(* CODESYS project Tc3_XPlanarStandard.library
   Company: Beckhoff Automation GmbH
   DefaultNamespace: Tc3_XPlanarStandard
   Version: 3.3.2411.0
   Placeholder: Tc3_XPlanarStandard
   Title: Tc3_XPlanarStandard

Project tree, tasks and I/O mapping:
  libraries: Tc2_EtherCAT, * (Beckhoff Automation GmbH); Tc2_Math, * (Beckhoff Automation GmbH); Tc2_MC2, * (Beckhoff Automation GmbH); Tc2_Standard, * (Beckhoff Automation GmbH); Tc2_System, * (Beckhoff Automation GmbH); Tc2_Utilities, * (Beckhoff Automation GmbH); Tc3_EventLogger, * (Beckhoff Automation GmbH); Tc3_Mc3PlanarMotion, * (Beckhoff Automation GmbH); Tc3_Module, * (Beckhoff Automation GmbH); Tc3_Physics, * (Beckhoff Automation GmbH); Tc3_XPlanarUtility, * (Beckhoff Automation GmbH)
  BaseMover/
    ITFs/
      interface I_MoverBase: MoverID
  GeneralStandardFunctions/
    function ConvertToEventEntry [ST]
    function block FB_TcMoverMessage [ST]: AddError, AddInfo, SendMessage, SetSucceeded
    data type ST_ActualMotionParameters
  Version/
    global variables Global_Version
  XPlanarStandardFunctions/
    JoinClosestTrack/
      DUTs/
        data type ST_ErrorDetails
        data type ST_TrackDistance
        data type ST_TrackReachingTrial
      function block FB_JoinClosestTrack [ST]: AddTrack, AssignMover, ClearTracks, Locked, TracksCount, Execute
    MotionSystem/
      DUTs/
        data type E_MethodKeepAliveMotionSystem
        data type ST_CommandReturn
        data type ST_CommandReturnGearInPosOnTrack
        data type ST_CommandReturnGearInPosOnTrackWithMasterMover
        data type ST_CommandReturnInfo
        data type ST_MoverCheckInfo
      function block FB_XPlanarSystem [ST]: P_AddEnviromentToGroup, P_AddModuleToEnvironment, P_AddMoversToGroup, P_AddMoverToGroup, P_AddTracksToGroup, P_CheckValidMovers, P_DisableGroup, P_DisableMovers, P_DisableTracks, P_EnableGroup, P_EnableMovers, P_EnableTrack, P_EnableTracks, P_HaltSystem, P_LeaveTrack, P_PartActivatePosition, P_PartAllowEnable, P_PartForceDisable, P_PartForceEnable, P_PartInitialize, P_PartInitializeMulti, P_PartReset, P_RemoveEnviromentFromGroup, P_RemoveMoverFromGroup, P_RemoveMoversFromGroup, P_RemoveTracksFromGroup, P_ResetGroup, P_ResetMovers, P_ResetParts, P_ResetTracks, AddEnvironmentToGroup, AddModuleToEnvironment, AddMoversToGroup, AddMoverToGroup, AddTracksToGroup, CheckValidMovers, DisableGroup, DisableMovers, DisableTracks, EnableGroup, EnableMovers, EnableTrack, EnableTracks, HaltSystem, LeaveTrack, PartActivatePosition, PartAllowEnable, PartForceDisable, PartForceEnable, PartInitialize, PartInitializeMulti, PartReset, RemoveEnvironmentFromGroup, RemoveMoverFromGroup, RemoveMoversFromGroup, RemoveTracksFromGroup, ResetGroup, ResetMovers, ResetParts, ResetTracks, UtilityCheckForError, UtilityErrorReset, ccl_AddEnvironmentToGroup, ccl_AddModuleToEnvironment, ccl_AddMoversToGroup, ccl_AddMoverToGroup, ccl_AddTracksToGroup, ccl_CheckValidMovers, ccl_DisableGroup, ccl_DisableMovers, ccl_DisableTracks, ccl_EnableGroup, ccl_EnableMovers, ccl_EnableTrack, ccl_EnableTracks, ccl_HaltSystem, ccl_LeaveTrack, ccl_MethodKeepAlive, ccl_PartActivatePosition, ccl_PartAllowEnable, ccl_PartForceDisable, ccl_PartForceEnable, ccl_PartInitialize, ccl_PartInitializeMulti, ccl_PartReset, ccl_RemoveEnvironmentFromGroup, ccl_RemoveMoverFromGroup, ccl_RemoveMoversFromGroup, ccl_RemoveTracksFromGroup, ccl_ResetGroup, ccl_ResetMovers, ccl_ResetParts, ccl_ResetTracks, ResetStateVariables, Cycle, ipDriver, ipTcIoMover, P_IndexXPU, P_SystemInitialized, SetMoverStandard, SetTrackStandard, WriteParameter
      interface I_MotionSystem: P_AddEnviromentToGroup, P_AddModuleToEnvironment, P_AddMoversToGroup, P_AddMoverToGroup, P_AddTracksToGroup, P_CheckValidMovers, P_DisableGroup, P_DisableMovers, P_DisableTracks, P_EnableGroup, P_EnableMovers, P_EnableTrack, P_EnableTracks, P_HaltSystem, P_LeaveTrack, P_PartActivatePosition, P_PartAllowEnable, P_PartForceDisable, P_PartInitialize, P_PartInitializeMulti, P_PartReset, P_RemoveEnviromentFromGroup, P_RemoveMoverFromGroup, P_RemoveMoversFromGroup, P_RemoveTracksFromGroup, P_ResetGroup, P_ResetMovers, P_ResetParts, P_ResetTracks, AddEnvironmentToGroup, AddModuleToEnvironment, AddMoversToGroup, AddMoverToGroup, AddTracksToGroup, CheckValidMovers, DisableGroup, DisableMovers, DisableTracks, EnableGroup, EnableMovers, EnableTrack, EnableTracks, HaltSystem, LeaveTrack, PartActivatePosition, PartAllowEnable, PartForceDisable, PartInitialize, PartInitializeMulti, PartReset, RemoveEnvironmentFromGroup, RemoveMoverFromGroup, RemoveMoversFromGroup, RemoveTracksFromGroup, ResetGroup, ResetMovers, ResetParts, ResetTracks, UtilityCheckForError, UtilityErrorReset, Cycle, ipDriver, P_IndexXPU, P_SystemInitialized, SetMoverStandard, SetTrackStandard, WriteParameter
    Mover/
      BaseFunctions/
        function MoverVectorToPostionXYC [ST]
      DUTs/
        Log/
          data type E_MoverCommandType
          data type ST_GearInPosOnTrackMasterMoverParameterLog
          data type ST_GearInPosOnTrackParameterLog
          data type ST_JoinTrackLog
          data type ST_LeaveTrackInPositionLog
          data type ST_LeaveTrackLog
          data type ST_MoveOnTrackParameters
          data type ST_MoveOnTrackParametersLog
          data type ST_MoverCommand
          data type ST_MoverCommandLog
          data type ST_MoveToPositionExtParametersLog
          data type ST_MoveToPositionParametersLog
          data type ST_SetPositionParametersLog
        data type E_HaltDynamicsMode
        data type ST_CheckStartConditionFeedback
        data type ST_CheckStartConditionFeedbackExt
        data type ST_DynamicsVADJ
        data type ST_HaltDynamics
        data type ST_HaltParameter
        data type ST_TrackTableInfo
      Experimental/
        function block FB_MoverTarget [ST]: AddMover, AddPosition, Clear, MoversToTarget, P_ErrorWarningCode, P_Info, SetDynamics
        data type ST_MoverDistance
      ITFs/
      function block FB_XPlanarMoverStandard [ST]: P_DcTimeStamp, GetCommandLog, MoverCommandToString, UpdateCommandHistory, CheckStartConditions, GetCustomTrackID, GetDistanceToTrack, GetLastKnownCustomTrackID, MoveOnTrack, MoveToPosition, AddToGroup, AdoptTrackOrientation, Disable, DisableExternalSetpointGeneration, Enable, EnableExternalSetpointGeneration, GearInPosOnTrack, GetPositionOnCurrentPart, Halt, JoinTrack, LeaveTrack, LeaveTrackInPosition, MoveA, MoveB, MoveC, MoveOnTrackExt, MoveToPositionExt, MoveToPositionXYC, MoveZ, RemoveFromGroup, Reset, SetExternalSetpointValues, SetMoverPosition, CopyReturnStructure, CopyReturnStructureGearInPosOnTrack, CopyReturnStructureGearInPosOnTrackMasterMover, UpdateActualMotionParameter, P_AtRotationPoint, P_ClosestQuaterAngle, P_CRotationRestrictions, P_CustomTrackIdTable, P_HaltDynamics, P_IsMovingXY, P_IsPresent, P_IsQueuing, P_IsSetpointGeneratorActive, P_LastKnownTrackOID, P_RotationAngleModulo, P_SavedMoveOnTrackParameter, P_ZeroVelocityThreshold, P_AddToGroup, P_AdoptTrackOrientation, P_Disable, P_DisableExternalSetpointGeneration, P_Enable, P_EnableExternalSetpointGeneration, P_GearInPosOnTrack, P_GearInPosOnTrackMasterMover, P_Halt, P_JoinTrack, P_LeaveTrack, P_LeaveTrackInPosition, P_MoveA, P_MoveB, P_MoveC, P_MoveOnTrack, P_MoveOnTrackExt, P_MoveToPosition, P_MoveToPositionExt, P_MoveToPositionXYC, P_MoveZ, P_RemoveFromGroup, P_Reset, P_SetMoverPosition, P_ActPosition, P_ActVelocity, P_Busy, P_CommandMode, P_Error, P_ErrorCode, P_ErrorID, P_Id, P_InGroup, P_MoverOid, P_MoverRef, P_PhysicalAreaID, P_SetAcceleration, P_SetOnTrack, P_SetPosition, P_SetVelocity, P_State, P_TrackId, Cycle
      interface I_XPlanarMoverStandard: P_DcTimeStamp, CheckStartConditions, GetCustomTrackID, GetDistanceToTrack, GetLastKnownCustomTrackID, MoveOnTrack, MoveToPosition, AddToGroup, AdoptTrackOrientation, Disable, DisableExternalSetpointGeneration, Enable, EnableExternalSetpointGeneration, GearInPosOnTrack, GetCommandLog, GetPositionOnCurrentPart, Halt, JoinTrack, LeaveTrack, LeaveTrackInPosition, MoveA, MoveB, MoveC, MoveOnTrackExt, MoveToPositionExt, MoveToPositionXYC, MoveZ, RemoveFromGroup, Reset, SetExternalSetpointValues, SetMoverPosition, P_AtRotationPoint, P_ClosestQuaterAngle, P_CRotationRestrictions, P_CustomTrackIdTable, P_HaltDynamics, P_IsMovingXY, P_IsPresent, P_IsQueuing, P_IsSetpointGeneratorActive, P_LastKnownTrackOID, P_RotationAngleModulo, P_SavedMoveOnTrackParameter, P_ZeroVelocityThreshold, P_AddToGroup, P_AdoptTrackOrientation, P_Disable, P_DisableExternalSetpointGeneration, P_Enable, P_EnableExternalSetpointGeneration, P_GearInPosOnTrack, P_GearInPosOnTrackMasterMover, P_Halt, P_JoinTrack, P_LeaveTrack, P_LeaveTrackInPosition, P_MoveA, P_MoveB, P_MoveC, P_MoveOnTrack, P_MoveOnTrackExt, P_MoveToPosition, P_MoveToPositionExt, P_MoveToPositionXYC, P_MoveZ, P_RemoveFromGroup, P_Reset, P_SetMoverPosition, P_ActPosition, P_ActVelocity, P_Busy, P_CommandMode, P_Error, P_ErrorCode, P_ErrorID, P_Id, P_InGroup, P_MoverOid, P_MoverRef, P_PhysicalAreaID, P_SetAcceleration, P_SetOnTrack, P_SetPosition, P_SetVelocity, P_State, P_TrackId, Cycle
    MoverQueue/
      DUTs/
        data type ST_MoverOnTrack
      function block FB_MoverQueue [ST]: Clear, Dequeue, Enqueue, Count, Item
      interface I_MoverQueue: Clear, Dequeue, Enqueue, Count, Item
    Station/
      DUTs/
        data type eSortingDirection
        data type eSortingMode
        data type ST_List
        data type ST_MoverInList
      function block FB_List [ST]: P_eSortingMode, P_fSortingOrigin, P_nNumberInList, P_nResult, P_nSortingMode, P_sMessage, P_SortingMode, AddMover, AddTrack, ClearList, ClearTrackOrder, CopyList, GetMoverIndexInListPosition, GetMoverInListPosition, P_FirstInList, P_Message, P_MoverList, P_NumberInList, P_Result, P_SortingDirection, P_SortingOrigin, P_TrackBuiltInfo, RemoveFirstInList, RemoveFromList, SortList
      interface I_List: P_eSortingMode, P_fSortingOrigin, P_nNumberInList, P_nResult, P_nSortingMode, P_sMessage, AddMover, AddTrack, ClearList, ClearTrackOrder, GetMoverIndexInListPosition, GetMoverInListPosition, P_FirstInList, P_Message, P_MoverList, P_NumberInList, P_Result, P_SortingMode, P_SortingOrigin, P_TrackBuiltInfo, RemoveFirstInList, RemoveFromList, SortList
    Track/
      DUTs/
        data type E_MethodKeepAliveTrack
        data type E_PointOption
        data type E_PointType
        data type E_TrackCommandType
        data type ST_BuildTrackParameterLog
        data type ST_CutomTrackID
        data type ST_LoggingVisu
        data type ST_StartEndAtTrackParameterLog
        data type ST_TrackAppendCircleParameterLog
        data type ST_TrackAppendLineParameterLog
        data type ST_TrackAppendPointParameterLog
        data type ST_TrackBuildParameter
        data type ST_TrackBuiltInfo
        data type ST_TrackCommand
        data type ST_TrackCommandLog
        data type ST_TrackInfo
        data type ST_TrackPoint
        data type ST_TrackTable
      function block FB_CustomTrackIdTable [ST]: Clear, P_TabelData, SetTrack
      function block FB_TrackStandard [ST]: ccl_BuildTrack, ccl_BuildTrackAdv, ccl_BuildTrackExt, ccl_MethodKeepAlive, CopyReturnStructure, ref, GetCommandLog, TrackCommandToString, UpdateCommandHistory, P_AddToGroup, P_AppendCircle, P_AppendLine, P_AppendPoint, P_BuildTrack, P_BuildTrackAdvanced, P_BuildTrackAdvanced_Check, P_BuildTrackAdvancedInfoText, P_BuildTrackExt, P_BuildTrackExtInfoText, P_Clear, P_CloseLoop, P_Disable, P_Enable, P_EndAtTrack, P_RemoveFromGroup, P_Reset, P_StartFromTrack, AddToGroup, AppendCircle, AppendLine, AppendPoint, BuildTrack, BuildTrackAdvanced, BuildTrackExt, Clear, CloseLoop, cycle, Disable, Enable, EndAtTrack, EndAtTrackAdv, GetLength, GetMoverPositionAt, GetTrackPositionAt, GetTrackPositionAt_XY, P_GroupOID, P_Info, P_MoverCountOnTrack, P_MovingMoverCount, P_OID, P_OperationMode, P_State, P_TrackBuiltInfo, P_TrackRef, RemoveFromGroup, Reset, StartFromTrack, StartFromTrackAdv
      function block FB_TrackTable [ST]: AddPoint, CheckTrackTable, ClearTrackTable, P_BuildlParameter, P_CloseTheLoop, P_EndAtTrack, P_InfoText, P_NumberOfPointsInTable, P_StartFromTrack, P_Table, P_TrackCheckImplausibleTableIndex, P_TrackTableCheckResult
      function block FB_TrackTableAdvanced [ST]: AddPoint, CheckPoint, CheckTrackTable, ClearTrackTable, P_BuildlParameter, P_CloseTheLoop, P_EndAtTrack, P_EndAtTrackOptions, P_InfoText, P_NumberOfPointsInTable, P_StartFromTrack, P_StartFromTrackOptions, P_Table, P_TrackCheckImplausibleTableIndex, P_TrackTableCheckResult
      interface I_CustomTrackIndexTable: P_TabelData
      interface I_TrackStandard: P_AddToGroup, P_AppendCircle, P_AppendLine, P_AppendPoint, P_BuildTrack, P_BuildTrackAdvanced, P_BuildTrackAdvanced_Check, P_BuildTrackAdvancedInfoText, P_BuildTrackExt, P_Clear, P_CloseLoop, P_Disable, P_Enable, P_EndAtTrack, P_RemoveFromGroup, P_Reset, P_StartFromTrack, AddToGroup, AppendCircle, AppendLine, AppendPoint, BuildTrack, BuildTrackAdvanced, BuildTrackExt, Clear, CloseLoop, Cycle, Disable, Enable, GetCommandLog, GetLength, GetMoverPositionAt, GetTrackPositionAt, GetTrackPositionAt_XY, P_GroupOID, P_Info, P_MoverCountOnTrack, P_MovingMoverCount, P_OID, P_OperationMode, P_State, P_TrackRef, ref, RemoveFromGroup, Reset
    Visualization/
      DUTs/
        data type ST_MoverVisualisation
        data type ST_TrackVisualisation
      Helper/
        visualisation VI_Background
      MoverLog/
        visualisation VI_MoverLogOverview
        visualisation VI_MoverLogOverview_Single
        visualisation VI_MoverLogOverview_Single_1
      TrackLog/
        visualisation VI_TrackLogOverview
        visualisation VI_TrackLogOverview_Single
      function block FB_XPlanarVisuDiag [ST]: Cycle, SetStandardMover, SetStandardTrack, UpdateMoverStatus, UpdateTrackLog
  text list GlobalTextList
  global variables GVL_internal
  global variables GVL_Tc3XPlanarStandard
  global variables Params_XPlanar
*)

// GeneralStandardFunctions/ST_ActualMotionParameters
TYPE ST_ActualMotionParameters :
STRUCT
	Position			: MoverVector;
	fSetTrackPosition	: LREAL;
	nTrackOid 			: OTCID;
	sTrackName 			: STRING(80);
	fSetVelo			: LREAL;
	fSetAcc				: LREAL;	
END_STRUCT
END_TYPE

// XPlanarStandardFunctions/JoinClosestTrack/DUTs/ST_ErrorDetails
TYPE ST_ErrorDetails :
STRUCT
	TrackOID	: OTCID;			// Track object ID
	ErrorID		: UDINT;			// Error ID
	objectInfo	: PlanarObjectInfo;	// Object causing error
END_STRUCT
END_TYPE

// XPlanarStandardFunctions/JoinClosestTrack/DUTs/ST_TrackDistance
TYPE ST_TrackDistance :
STRUCT
	TrackOID		: OTCID;			// Track object ID
	Index			: UDINT;			// Index in Track list
	CurrentLocation	: MoverVector;		// Current position of the Mover
	PositionOnTrack	: LREAL;			// Arc position on Track after JoinTrack() command
	IsPossibleTrack	: BOOL;				// Joining this track is possible
	ErrorID			: UDINT;			// Error ID making track impossible to join
	objectInfo		: PlanarObjectInfo;	// Object causing collision
	TargetLocation	: MoverVector;		// Mover position after JoinTrack() command
	Distance		: LREAL;			// Absolute distance [mm]
END_STRUCT
END_TYPE

// XPlanarStandardFunctions/JoinClosestTrack/DUTs/ST_TrackReachingTrial
TYPE ST_TrackReachingTrial :
STRUCT
	TrackInfo	: ST_TrackDistance;	// Track distance info
	Done		: BOOL;				// JoinTrack operation has succeed
	Busy		: BOOL;				// JoinTrack operation is busy
	Error		: BOOL;				// JoinTrack operation has failed
	ErrorID		: UDINT;			// Error ID at failure
	objectInfo	: PlanarObjectInfo;	// Object causing collision
END_STRUCT
END_TYPE

// XPlanarStandardFunctions/MotionSystem/DUTs/E_MethodKeepAliveMotionSystem
{attribute 'qualified_only'}
{attribute 'strict'}
TYPE E_MethodKeepAliveMotionSystem :
(
	eIdle := 0,
	eAddMoverToGroup,
	eAddMoversToGroup,
	eAddEnvironmentToGroup,
	eAddTracksToGroup,
	eDisableGroup,
	eDisableMovers,
	eDisableSystem,
	eEnableGroup,
	eEnableMovers,
	eEnableSystem,
	eEnableTrack,
	eEnableTracks,
	eDisableTracks,
	eHaltSystem,
	eLeaveTrack,
	eRemoveMoverFromGroup,
	eRemoveMoversFromGroup,
	eRemoveEnvironmentFromGroup,
	eRemoveTracksFromGroup,
	eResetGroup,
	eResetTracks,
	eResetMovers,
	eResetSystem,
	eError,
	eAddModuleToEnvironment,
	eCheckValidMovers,
	ePartInitialize,
	ePartInitializeMulti,
	ePartActivatePosition,
	ePartForceDisable,
	ePartForceEnable,
	ePartAllowEnable,
	ePartReset,
	eResetParts
);
END_TYPE

// XPlanarStandardFunctions/MotionSystem/DUTs/ST_CommandReturn
TYPE ST_CommandReturn :
STRUCT
	Done 	: BOOL;
	Busy 	: BOOL;
	Aborted	: BOOL;
	Active 	: BOOL;
	Error	: BOOL;
	ErrorID	: UDINT;
	stInfo 	: ST_CommandReturnInfo;
END_STRUCT
END_TYPE

// XPlanarStandardFunctions/MotionSystem/DUTs/ST_CommandReturnGearInPosOnTrack
TYPE ST_CommandReturnGearInPosOnTrack :
STRUCT
//	Done 	: BOOL;
	Busy 	: BOOL;
	Aborted	: BOOL;
	Active 	: BOOL;
	Error	: BOOL;
	ErrorID	: UDINT;
	stInfo 	: ST_CommandReturnInfo;
	inSync	: BOOL;
END_STRUCT
END_TYPE

// XPlanarStandardFunctions/MotionSystem/DUTs/ST_CommandReturnGearInPosOnTrackWithMasterMover
TYPE ST_CommandReturnGearInPosOnTrackWithMasterMover :
STRUCT
//	Done 	: BOOL;
	Busy 	: BOOL;
	Aborted	: BOOL;
	Active 	: BOOL;
	Error	: BOOL;
	ErrorID	: UDINT;
	stInfo 	: ST_CommandReturnInfo;
	inSync	: BOOL;
END_STRUCT
END_TYPE

// XPlanarStandardFunctions/MotionSystem/DUTs/ST_CommandReturnInfo
TYPE ST_CommandReturnInfo :
STRUCT
	nObjectType : UDINT;
	nObjectID 	: UDINT;
END_STRUCT
END_TYPE

// XPlanarStandardFunctions/MotionSystem/DUTs/ST_MoverCheckInfo
TYPE ST_MoverCheckInfo :
STRUCT
	bDone				: BOOL;	
	bAllMoversValid		: BOOL;
	bMoverLost			: BOOL;
	nValidMoverCount	: UDINT;	

END_STRUCT
END_TYPE

// XPlanarStandardFunctions/Mover/DUTs/Log/E_MoverCommandType
TYPE E_MoverCommandType :
(
	eMoverCommand_eNoCommand 			:= 0,
	eMoverCommand_eMoveAbs,
	eMoverCommand_eMoveModOnTrack,
	eMoverCommand_eMoveModOnTrackExt,		
	eMoverCommand_eMoveRel,			
	eMoverCommand_eHalt, 			
	eMoverCommand_eGearIn, 			
	eMoverCommand_eDynamicsChange, 		
	eMoverCommand_eGapChange, 		
	eMoverCommand_eSuperImposed, 	
	eMoverCommand_eCamInInstant, 	
	eMoverCommand_eCamInTwoTables, 	
	eMoverCommand_eCamOut, 			
	eMoverCommand_eReset, 			
	eMoverCommand_eEnable,			
	eMoverCommand_eDisable,			
	eMoverCommand_eAddMoverToGroup,	
	eMoverCommand_eRemoveMoverFromGroup,	
	eMoverCommand_eMoveAbsDone,		
	eMoverCommand_eMoveModDone,		
	eMoverCommand_eMoveRelDone,			
	eMoverCommand_eHaltCa,				
	eMoverCommand_eHaltCaDone,			
	eMoverCommand_eMoveAbsQueueing,	
	eMoverCommand_eMoveModQueueing,		
	eMoverCommand_eMoveRelQueueing,		
	eMoverCommand_eGearInInSync,		
	eMoverCommand_eGearOutOfSync,	
	eMoverCommand_eJoinTrack,			
	eMoverCommand_eLeaveTrack,		
	eMoverCommand_eLeaveTrackInPosition,	
	eMoverCommand_eMoveToPosition,		
	eMoverCommand_eMoveToPositionXYC,	
	eMoverCommand_eMoveToPositionExt,	
	eMoverCommand_eMoveZ,
	eMoverCommand_eMoveA,
	eMoverCommand_eMoveB,
	eMoverCommand_eMoveC,
	eMoverCommand_eEnableExternalSetPos,
	eMoverCommand_eDisableExternalSetPos,
	eMoverCommand_eCheckStartConditions,
	eMoverCommand_eAdoptTrackOrientation,
	eMoverCommand_eGearInPosOnTrack,
	eMoverCommand_eGearInPosOnTrackMasterMover,
	eMoverCommand_eSetPosition 	
	
	
);
END_TYPE

// XPlanarStandardFunctions/Mover/DUTs/Log/ST_GearInPosOnTrackMasterMoverParameterLog
TYPE ST_GearInPosOnTrackMasterMoverParameterLog :
STRUCT
	
	MasterMover			: UDINT;
	MasterSyncPos		: LREAL;
	TrackMasterSyncPos	: UDINT;
	SlaveSyncPos		: LREAL;
	TrackSlaveSyncPos	: UDINT;
	
	TrackTrailSize		: UDINT;	
	
	Velocity  			: LREAL;
	Acceleration		: LREAL;
	Deceleration		: LREAL;
	Jerk  				: LREAL;
	Gap					: LREAL;

	moduloToleranceMasterSyncPosition	: LREAL;
	directionMasterSyncPosition			: DINT;
	inSyncToleranceDistance				: LREAL;
	moduloToleranceSlaveSyncPosition	: LREAL;
	
	allowedSlaveSyncDirections			: DINT;
	directionSlaveSyncPosition			: DINT;
	
	followMover							: BOOL;
	
	
	

		
END_STRUCT
END_TYPE

// XPlanarStandardFunctions/Mover/DUTs/Log/ST_GearInPosOnTrackParameterLog
TYPE ST_GearInPosOnTrackParameterLog :
STRUCT
	
	MasterSyncPos	: LREAL;
	SlaveSyncPos	: LREAL;
	Velocity  		: LREAL;
	Acceleration	: LREAL;
	Deceleration	: LREAL;
	Jerk  			: LREAL;
	Gap				: LREAL;

	Track			: UDINT;
	TrackTrailSize	: UDINT;
	
	allowedSlaveSyncDirections	: Tc3_Mc3PlanarMotion.MC_SYNC_DIRECTIONS;
	directionSlaveSyncPosition  : Tc3_Mc3PlanarMotion.MC_Direction;
	
	inSyncToleranceDistance				: LREAL;
	moduloToleranceSlaveSyncPosition	: LREAL;
	
		
END_STRUCT
END_TYPE

// XPlanarStandardFunctions/Mover/DUTs/Log/ST_JoinTrackLog
TYPE ST_JoinTrackLog :
STRUCT
	nTargetTrack 		: OTCID;
	fVelo				: LREAL;		
	fAcc				: LREAL;
	fJerk				: LREAL;
END_STRUCT
END_TYPE

// XPlanarStandardFunctions/Mover/DUTs/Log/ST_LeaveTrackInPositionLog
TYPE ST_LeaveTrackInPositionLog :
STRUCT
	fPositionX			: LREAL;		
	fPositionY			: LREAL;		
	fPositionC			: LREAL;		
END_STRUCT
END_TYPE

// XPlanarStandardFunctions/Mover/DUTs/Log/ST_LeaveTrackLog
TYPE ST_LeaveTrackLog :
STRUCT
	fPositionX			: LREAL;		
	fPositionY			: LREAL;		
	fPositionC			: LREAL;		
	fVelo				: LREAL;		
	fAcc				: LREAL;
	fDec				: LREAL;
	fJerk				: LREAL;
END_STRUCT
END_TYPE

// XPlanarStandardFunctions/Mover/DUTs/Log/ST_MoveOnTrackParameters
TYPE ST_MoveOnTrackParameters:
STRUCT
	
	fTrackPosition	 	: LREAL;
	fVelo				: LREAL;	
	ipTrack				: I_TrackStandard;
	fAcc				: LREAL;
	fDec				: LREAL;
	fJerk				: LREAL;
	fGap				: LREAL;
	direction			: Tc3_Mc3PlanarMotion.MC_DIRECTION;
	
END_STRUCT
END_TYPE

// XPlanarStandardFunctions/Mover/DUTs/Log/ST_MoveOnTrackParametersLog
TYPE ST_MoveOnTrackParametersLog:
STRUCT
	
	fTargetPosition 	: LREAL;
	fVelo				: LREAL;	
	nTargetTrackOid		: OTCID;
	sTargetTrack		: STRING(80);
	nTargetTrackID		: UDINT;
	fAcc				: LREAL;
	fDec				: LREAL;
	fJerk				: LREAL;
	fGap				: LREAL;
	
END_STRUCT
END_TYPE

// XPlanarStandardFunctions/Mover/DUTs/Log/ST_MoverCommand
TYPE ST_MoverCommand : //structure for storing a list of commands to the mover 
STRUCT
	sStation				: STRING;	// Station Name that give a move command
	eCommandType 			: E_MoverCommandType; // what command was done
	
	stActualParameter			: ST_ActualMotionParameters;
//	stActualMasterParameter	: ST_ActualMotionParameters;
//	stGearInParameter		: ST_GearInParametersLog;
//	stMoveAbsoluteParameter	: ST_MoveAbsoluteParametersLog;
//	stMoveRelativeParameter	: ST_MoveRelativeParametersLog;
	stMoveOnTrackParameter					: ST_MoveOnTrackParametersLog;	
	stMoveOnTrackParameterExt				: ST_MoveOnTrackParametersLog;	
	stGearInPosOnTrackParameter				: ST_GearInPosOnTrackParameterLog;
	stGearInPosOnTrackMasterMoverParameter	: ST_GearInPosOnTrackMasteRMoverParameterLog;
	stMoveToPosition						: ST_MoveToPositionParametersLog;
	stMoveToPositionXYC						: ST_MoveToPositionParametersLog;
	stMoveToPositionExt						: ST_MoveToPositionExtParametersLog;	
 	stHaltParameter							: ST_HaltParameter;
	stJoinTrackParameter					: ST_JoinTrackLog;
	stLeaveTrackParameter					: ST_LeaveTrackLog;
	stLeaveTrackInPositionParameter			: ST_LeaveTrackInPositionLog;
	stSetPosition							: ST_SetPositionParametersLog;

	
	sText 					: STRING(255); 
	stTimeStamp 			: STRING ; //dcTimestampTime can be decoded later 
END_STRUCT
END_TYPE

// XPlanarStandardFunctions/Mover/DUTs/Log/ST_MoverCommandLog
TYPE ST_MoverCommandLog :
STRUCT
	nNo				: INT;
	sTimeStamp		: STRING;	
	sTimeStampDate	: STRING;
	sTimeStampTime	: STRING;	
	sStation		: STRING;
	sCommandType	: STRING;
	sText			: STRING(255);
END_STRUCT
END_TYPE

// XPlanarStandardFunctions/Mover/DUTs/Log/ST_MoveToPositionExtParametersLog
TYPE ST_MoveToPositionExtParametersLog:
STRUCT
	fVelo						: LREAL;	

	fTargetPositionX 			: LREAL;
	fTargetPositionY 			: LREAL;
	fTargetPositionC 			: LREAL;
	
	fAcc						: LREAL;
	fDec						: LREAL;
	fJerk						: LREAL;
	
	stMoveToPositionOptions		: ST_MoveToPositionOptions;
END_STRUCT
END_TYPE

// XPlanarStandardFunctions/Mover/DUTs/Log/ST_MoveToPositionParametersLog
TYPE ST_MoveToPositionParametersLog:
STRUCT


	fVelo				: LREAL;	

	fTargetPositionX 	: LREAL;
	fTargetPositionY 	: LREAL;
	fTargetPositionC 	: LREAL;
	
	fAcc				: LREAL;
	fDec				: LREAL;
	fJerk				: LREAL;	
	
	
END_STRUCT
END_TYPE

// XPlanarStandardFunctions/Mover/DUTs/Log/ST_SetPositionParametersLog
TYPE ST_SetPositionParametersLog:
STRUCT
	fPositionX 	: LREAL;
	fPositionY 	: LREAL;
	fPositionC 	: LREAL;
END_STRUCT
END_TYPE

// XPlanarStandardFunctions/Mover/DUTs/E_HaltDynamicsMode
{attribute 'qualified_only'}
{attribute 'strict'}
TYPE E_HaltDynamicsMode :
(
	AxisX_AxisY_CoordinatedOnPath 	:= 0,
	AxisX_AxisY_Separately			:= 1
);
END_TYPE

// XPlanarStandardFunctions/Mover/DUTs/ST_CheckStartConditionFeedback
TYPE ST_CheckStartConditionFeedback :
STRUCT

	nMoverID					: UINT;
	bPositionOK					: BOOL;	
	bPositionXLimitExceeded		: BOOL;
	bPositionYLimitExceeded		: BOOL;
	bAngleLimitExceeded			: BOOL;
	fCurrentAngleDeviation		: LREAL;
	fCurrentPositionDeviationX	: LREAL;
	fCurrentPositionDeviationY	: LREAL;	
	
END_STRUCT
END_TYPE

// XPlanarStandardFunctions/Mover/DUTs/ST_CheckStartConditionFeedbackExt
TYPE ST_CheckStartConditionFeedbackExt :
STRUCT

	nMoverID					: UINT;
	bPositionOK					: BOOL;	
	bFeedbackInvalid			: BOOL;
	bPositionXLimitExceeded		: BOOL;
	bPositionYLimitExceeded		: BOOL;
	bAngleLimitExceeded			: BOOL;
	fCurrentAngleDeviation		: LREAL;
	fCurrentPositionDeviationX	: LREAL;
	fCurrentPositionDeviationY	: LREAL;	
	
END_STRUCT
END_TYPE

// XPlanarStandardFunctions/Mover/DUTs/ST_DynamicsVADJ
TYPE ST_DynamicsVADJ :
STRUCT
	fVelocity		: LREAL;
	fAcceleration	: LREAL;
	fDeceleration	: LREAL;
	fJerk			: LREAL;	
END_STRUCT
END_TYPE

// XPlanarStandardFunctions/Mover/DUTs/ST_HaltDynamics
TYPE ST_HaltDynamics :
STRUCT
	
	PathXY		: ST_DynamicsVADJ;
	AxisX		: ST_DynamicsVADJ;
	AxisY		: ST_DynamicsVADJ;
	AxisZ		: ST_DynamicsVADJ;
	AxisA		: ST_DynamicsVADJ;
	AxisB		: ST_DynamicsVADJ;
	AxisC		: ST_DynamicsVADJ;	
	
	Mode		: E_HaltDynamicsMode;

END_STRUCT
END_TYPE

// XPlanarStandardFunctions/Mover/DUTs/ST_HaltParameter
TYPE ST_HaltParameter :
STRUCT
	
	fDeceleration_XY	: LREAL;
	fJerk_XY			: LREAL; 
	fDeceleration_A		: LREAL;
	fJerk_A				: LREAL; 
	fDeceleration_B		: LREAL;
	fJerk_B				: LREAL; 		
	fDeceleration_C		: LREAL;
	fJerk_C				: LREAL; 	
	
END_STRUCT
END_TYPE

// XPlanarStandardFunctions/Mover/DUTs/ST_TrackTableInfo
TYPE ST_TrackTableInfo :
STRUCT
	nTrackOID	: UDINT;
	nTrackID	: UDINT;	
END_STRUCT
END_TYPE

// XPlanarStandardFunctions/Mover/Experimental/ST_MoverDistance
{attribute 'hide'}
TYPE ST_MoverDistance :
STRUCT
	nPositionIndex	: UDINT;
	fDistance		: LREAL;
END_STRUCT
END_TYPE

// XPlanarStandardFunctions/MoverQueue/DUTs/ST_MoverOnTrack
TYPE ST_MoverOnTrack :
STRUCT
	ID			: UDINT;	// Mover ID
	MoverOID	: OTCID;	// Mover object ID
	PosOnTrack	: LREAL;	// Position on track
END_STRUCT
END_TYPE

// XPlanarStandardFunctions/Station/DUTs/eSortingDirection
TYPE eSortingDirection :
(
	ascending  := 0,
	descending := 1
);
END_TYPE

// XPlanarStandardFunctions/Station/DUTs/eSortingMode

TYPE eSortingMode :
(
	descending := 0,
	ascending  := 1
);
END_TYPE

// XPlanarStandardFunctions/Station/DUTs/ST_List
TYPE ST_List :
STRUCT
	nNumInList		: INT;
	//aMoverList 		: ARRAY[1..GVL_ListParameter.gcnMaxNumInList] OF I_XPlanarMoverStandard; 
	aMoverList 		: ARRAY[1..maxNumMover] OF I_XPlanarMoverStandard;
	
END_STRUCT
END_TYPE

// XPlanarStandardFunctions/Station/DUTs/ST_MoverInList
TYPE ST_MoverInList :
STRUCT
	nMoverIndex		 	: UDINT;
	nMoverPosition 		: LREAL;
	nMoverTrackOID 		: UDINT;	
END_STRUCT
END_TYPE

// XPlanarStandardFunctions/Track/DUTs/E_MethodKeepAliveTrack
{attribute 'qualified_only'}
{attribute 'strict'}
TYPE E_MethodKeepAliveTrack :
(
	eIdle          := 0,
	eBuildTrack    := 1,
	eBuildTrackExt := 2,
	eBuildTrackAdv := 3,
	eError
);
END_TYPE

// XPlanarStandardFunctions/Track/DUTs/E_PointOption
{attribute 'qualified_only'}
{attribute 'strict'}
TYPE E_PointOption :
(
	none,
	Circle_Clockwise,
	Circle_CounterClockwise
);
END_TYPE

// XPlanarStandardFunctions/Track/DUTs/E_PointType
{attribute 'qualified_only'}
{attribute 'strict'}
TYPE E_PointType :
(
	none,
	Point,
	Line_Start,
	Line_End,
	Circle_Start,
	Circle_Center,
	Circle_End
	
);
END_TYPE

// XPlanarStandardFunctions/Track/DUTs/E_TrackCommandType
TYPE E_TrackCommandType :
(
	eTrackCommand_eNoCommand 			:= 0,
	eTrackCommand_eEnable				:= 1,
	eTrackCommand_eDisable 				:= 2,
	eTrackCommand_eAppendLine 			:= 3,
	eTrackCommand_eCloseLoop			:= 4,
	eTrackCommand_eStartFromTrack		:= 5,	
	eTrackCommand_eEndAtTrack			:= 6,
	eTrackCommand_eAddToGroup			:= 7,
	eTrackCommand_eRemoveFromGroup		:= 8,
	eTrackCommand_eAppendPoint			:= 9,
	eTrackCommand_eAppendCircle			:= 10,
	eTrackCommand_eBuildTrack			:= 11,	
	eTrackCommand_eReset				:= 12,
	eTrackCommand_eClear				:= 13,
	eTrackCommand_eStartFromTrackAdv	:= 14,
	eTrackCommand_eAppendPointAdv		:= 15,
	eTrackCommand_eAppendLineAdv		:= 16,
	eTrackCommand_eAppendCircleAdv		:= 17
	
);
END_TYPE

// XPlanarStandardFunctions/Track/DUTs/ST_BuildTrackParameterLog
TYPE ST_BuildTrackParameterLog :
STRUCT
	
	bSuccess		: BOOL;
	bError			: BOOL;
	nErrorCode		: UDINT;
	fTrackLength	: LREAL;
	sBuildInfoText	: STRING;

END_STRUCT
END_TYPE

// XPlanarStandardFunctions/Track/DUTs/ST_CutomTrackID
TYPE ST_CutomTrackID :
STRUCT
	
	TrackOID	: OTCID;
	nCustomID	: UDINT;		

END_STRUCT
END_TYPE

// XPlanarStandardFunctions/Track/DUTs/ST_LoggingVisu
TYPE ST_LoggingVisu :
STRUCT
	
	nScrollBarMin 	: UINT;
	nScrollBarMax	: UINT;
	nScrollBarValue	: UINT;

END_STRUCT
END_TYPE

// XPlanarStandardFunctions/Track/DUTs/ST_StartEndAtTrackParameterLog
TYPE ST_StartEndAtTrackParameterLog :
STRUCT
	nTrackOID	: UDINT;	

END_STRUCT
END_TYPE

// XPlanarStandardFunctions/Track/DUTs/ST_TrackAppendCircleParameterLog
TYPE ST_TrackAppendCircleParameterLog:
	STRUCT
	startPositionX	:  LREAL;
	startPositionY	:  LREAL;
	
	centerPositionX	: LREAL;
	centerPositionY	: LREAL;
	
	endPositionX 	:  LREAL;
	endPositionY 	:  LREAL;
	END_STRUCT
END_TYPE

// XPlanarStandardFunctions/Track/DUTs/ST_TrackAppendLineParameterLog
TYPE ST_TrackAppendLineParameterLog:
	STRUCT
	startPositionX	:  LREAL;
	startPositionY	:  LREAL;
	
	
	endPositionX 	:  LREAL;
	endPositionY 	:  LREAL;
	END_STRUCT
END_TYPE

// XPlanarStandardFunctions/Track/DUTs/ST_TrackAppendPointParameterLog
TYPE ST_TrackAppendPointParameterLog:
	STRUCT
	positionX	:  LREAL;
	positionY 	:  LREAL;
	END_STRUCT
END_TYPE

// XPlanarStandardFunctions/Track/DUTs/ST_TrackBuildParameter
TYPE ST_TrackBuildParameter :
STRUCT
	StartFromTrack 	: I_TrackStandard;	
	EndAtTrack		: I_TrackStandard;	
	bCloseTheLoop	: BOOL;
	
	startOptions	: ST_StartFromTrackAdvancedOptions;
	endOptions		: ST_EndAtTrackAdvancedOptions;

END_STRUCT
END_TYPE

// XPlanarStandardFunctions/Track/DUTs/ST_TrackBuiltInfo
TYPE ST_TrackBuiltInfo :
STRUCT
	nTrackBuiltCountInfo	: UDINT;
	TrackInfo				: ARRAY[1..maxTrackCount] OF ST_TrackInfo;	
END_STRUCT
END_TYPE

// XPlanarStandardFunctions/Track/DUTs/ST_TrackCommand
TYPE ST_TrackCommand :
STRUCT
	eCommandType 			: E_TrackCommandType; // what command was done

	stTrackAppendLine		: ST_TrackAppendLineParameterLog;
	stTrackAppendPoint		: ST_TrackAppendPointParameterLog;
	stTrackAppendCircle		: ST_TrackAppendCircleParameterLog;
	stBuildTrack			: ST_BuildTrackParameterLog;
	stEndAtTrack			: ST_StartEndAtTrackParameterLog;
	stStartFromTrack		: ST_StartEndAtTrackParameterLog;
	
	sText 					: STRING(255); 
	stTimeStamp 			: STRING ; //dcTimestampTime can be decoded later 	
END_STRUCT
END_TYPE

// XPlanarStandardFunctions/Track/DUTs/ST_TrackCommandLog
TYPE ST_TrackCommandLog :
STRUCT
	nNo				: INT;
	sTimeStamp		: STRING;
	sTimeStampDate	: STRING;	
	sTimeStampTime	: STRING;
	sCommandType	: STRING;
	sText			: STRING(255);
END_STRUCT
END_TYPE

// XPlanarStandardFunctions/Track/DUTs/ST_TrackInfo
TYPE ST_TrackInfo :
STRUCT
	
	TrackOID		: UDINT;
	StartFromTrack	: I_TrackStandard;
	EndAtTrack		: I_TrackStandard;
	
END_STRUCT
END_TYPE

// XPlanarStandardFunctions/Track/DUTs/ST_TrackPoint
TYPE ST_TrackPoint :
STRUCT
	ePointType		: E_PointType;
	eOption			: E_PointOption;
	Position_X		: LREAL;
	Position_Y		: LREAL;
	Orientation_C	: LREAL;	
END_STRUCT
END_TYPE

// XPlanarStandardFunctions/Track/DUTs/ST_TrackTable
TYPE ST_TrackTable :
STRUCT
	
	fPointPosition_X		: LREAL;
	fPointPosition_Y		: LREAL;
	fPointOrientation_C		: LREAL;
	ePointType				: E_PointType;
	eOption					: E_PointOption;
	ReferenceSystem			: OTCID;

END_STRUCT
END_TYPE

// XPlanarStandardFunctions/Visualization/DUTs/ST_MoverVisualisation
TYPE ST_MoverVisualisation :
STRUCT
	stMoverPos : MoverVector;
	stMoverVelo: MoverVector;
	stMoverAcc : MoverVector;
	
	nID			: UDINT;
	trackPos	: LREAL;
	bError		: BOOL;
	nErrorID	: UDINT;
	
	eState 				: MC_PLANAR_STATE;
	eActivationState	: MC_PLANAR_MOVER_COMMAND_MODE;
	
	bBusy		: BOOL;
	bActivated 	: BOOL;
	bOnTrack	: BOOL;
	bActivating : BOOL;
	bInactive	: BOOL;
END_STRUCT
END_TYPE

// XPlanarStandardFunctions/Visualization/DUTs/ST_TrackVisualisation
TYPE ST_TrackVisualisation :
STRUCT

END_STRUCT
END_TYPE

// Version/Global_Version
{attribute 'TcGenerated'}
{attribute 'no-analysis'}
{attribute 'linkalways'}
// This function has been automatically generated from the project information.
VAR_GLOBAL CONSTANT
	{attribute 'const_non_replaced'}
	stLibVersion_Tc3_XPlanarStandard : ST_LibVersion := (iMajor := 3, iMinor := 3, iBuild := 2411, iRevision := 0, nFlags := 0, sVersion := '3.3.2411.0');
END_VAR

// GVL_internal
{attribute 'qualified_only'}
VAR_GLOBAL
	{attribute 'hide'}


	// Mover log
	nMoverIdToDisplay 		: INT := 1;	
	//nMaxMoverIdtoDisplay 	: INT := 10;
	bPreviousMover			: BOOL;
	bNextMover				: BOOL;
	//rTrigNextMover			: R_TRIG;
	//rTirgPreviousMover		: R_TRIG;
	stMoverCmdLog 			: ARRAY [1..10] OF ST_MoverCommandLog;
	stMoverVisuData			: ST_LoggingVisu;

	// Track log	
	nTrackIdToDisplay 		: INT := 1;	
	//nMaxTrackIdtoDisplay 	: INT := 10;
	bPreviousTrack			: BOOL;
	bNextTrack				: BOOL;
	//rTrigNextTrack			: R_TRIG;
	//rTirgPreviousTrack		: R_TRIG;
	stTrackCmdLog 			: ARRAY [1..10] OF ST_TrackCommandLog;
	stTrackVisuData			: ST_LoggingVisu;	

	

END_VAR



(*
VAR_GLOBAL CONSTANT
	gcnMaxStation			: INT := 10;
	gcnMaxMoverInStation	: INT := 20;
END_VAR
*)

// GVL_Tc3XPlanarStandard
VAR_GLOBAL
	fbEnvironment			: FB_TcIoXPlanarEnvironment;
	fbTcIoXPlanarMover		: ARRAY [1..Params_XPlanar.maxNumMover] OF FB_TcIoXPlanarMover;
	fbTcIoXPlanarTile		: ARRAY [1..Param_TcIoXplanarEnvironment.MaxTiles] OF FB_TcIoXPlanarTile;
	fbVisuXPlanarDiag		: FB_XPlanarUtilityVisu;
	fbXPlanarVisuDiag		: FB_XPlanarVisuDiag;
END_VAR

// Params_XPlanar

VAR_GLOBAL CONSTANT
	
	moverCount			: UDINT := 4;
	MAX_LAST_LOGS		: UINT  := 25;
	maxNumTrackPoints	: UINT  := 20;
	maxTrackCount		: UDINT := 10;
	maxNumStation		: UDINT := 3;
	maxNumMover 		: UDINT := 20;
	maxNumberOfParts	: UDINT := 20;
	
END_VAR

// BaseMover/ITFs/I_MoverBase
INTERFACE I_MoverBase

PROPERTY MoverID : INT
GET
END_GET
SET
END_SET
END_PROPERTY

END_INTERFACE

// GeneralStandardFunctions/ConvertToEventEntry
FUNCTION ConvertToEventEntry : TcEventEntry
VAR_INPUT
	nEventId 		: UDINT;
	uuidEventClass 	: GUID;
END_VAR

ConvertToEventEntry.uuidEventClass 	:= uuidEventClass;
ConvertToEventEntry.nEventId 		:= nEventId;

END_FUNCTION

// GeneralStandardFunctions/FB_TcMoverMessage
FUNCTION_BLOCK FB_TcMoverMessage EXTENDS FB_TcMessage 
VAR_INPUT
END_VAR
VAR_OUTPUT
END_VAR
VAR
	fbSource	: FB_TcSourceInfo;
END_VAR

METHOD AddError : BOOL
VAR_INPUT
	nEventId 		: UDINT;
	uuidEventClass 	: GUID;
	ExtendSource	: STRING; 
END_VAR
VAR
	eventEntry : Tc3_EventLogger.TcEventEntry;
END_VAR
eventEntry := ConvertToEventEntry(nEventId, uuidEventClass);
eventEntry.eSeverity := TcEventSeverity.Error;
fbSource.ResetToDefault();
IF ExtendSource <> '' THEN
	fbSource.ExtendName('.');
	fbSource.ExtendName(ExtendSource);
END_IF
IF NOT THIS^.EqualsToEventEntryEx(stOther := eventEntry) THEN	
	THIS^.CreateEx(eventEntry, fbSource);
	THIS^.Send(0);
END_IF
END_METHOD

METHOD AddInfo : HRESULT
VAR_INPUT
	nEventId 		: UDINT;
	uuidEventClass 	: GUID;
	ExtendSource	: STRING; 
END_VAR
VAR
	eventEntry : Tc3_EventLogger.TcEventEntry;
END_VAR
eventEntry := ConvertToEventEntry(nEventId, uuidEventClass);
eventEntry.eSeverity := TcEventSeverity.Info;
fbSource.ResetToDefault();
IF ExtendSource <> '' THEN
	fbSource.ExtendName('.');
	fbSource.ExtendName(ExtendSource);
END_IF
IF NOT THIS^.EqualsToEventEntryEx(stOther := eventEntry) THEN	
	THIS^.CreateEx(eventEntry, 0);
	THIS^.Send(0);
END_IF
END_METHOD

METHOD SendMessage : HRESULT
VAR_INPUT
	eventEntry					: TcEventEntry;
	uuidEventClass 				: GUID;
	stCommand 					: ST_MoverCommand;
	stActualMotionParameter		: ST_ActualMotionParameters;	
END_VAR

VAR_INST
	hresult : HRESULT;
END_VAR
THIS^.CreateEx(eventEntry, 0);
CASE stCommand.eCommandType OF	
(*	eMoverCommand_eMoveABS:	
		THIS^.ipArguments.Clear();	
		THIS^.ipArguments.AddString(stCommand.sText);									//0
		THIS^.ipArguments.AddString(stCommand.sStation);								//1
		THIS^.ipArguments.AddLReal(stActualMotionParameter.fSetModuloPosition);			//2
		THIS^.ipArguments.AddLReal(stActualMotionParameter.fSetPosition);				//3
		THIS^.ipArguments.AddLReal(stActualMotionParameter.fSetVelo);					//4
		THIS^.ipArguments.AddLReal(stActualMotionParameter.fSetAcc);					//5
		THIS^.ipArguments.AddLReal(stCommand.stMoveAbsoluteParameter.fPosition);		//6
		THIS^.ipArguments.AddLReal(stCommand.stMoveAbsoluteParameter.fVelocity);		//7
		THIS^.ipArguments.AddLReal(stCommand.stMoveAbsoluteParameter.fAccel);			//8
		THIS^.ipArguments.AddLReal(stCommand.stMoveAbsoluteParameter.fDecel);			//9
		THIS^.ipArguments.AddLReal(stCommand.stMoveAbsoluteParameter.fJerk);			//10
		THIS^.ipArguments.AddLReal(stCommand.stMoveAbsoluteParameter.fGap);				//11
						
	eMoverCommand_eMoveMOD :
		THIS^.ipArguments.Clear();													
		THIS^.ipArguments.AddString(stCommand.sText);										//0
		THIS^.ipArguments.AddString(stCommand.sStation);									//1
		THIS^.ipArguments.AddLReal(stActualMotionParameter.fSetModuloPosition);				//2
		THIS^.ipArguments.AddLReal(stActualMotionParameter.fSetPosition);					//3
		THIS^.ipArguments.AddLReal(stActualMotionParameter.fSetVelo);						//4
		THIS^.ipArguments.AddLReal(stActualMotionParameter.fSetAcc);						//5
		THIS^.ipArguments.AddLReal(stCommand.stMoveModuloParameter.fPosition);				//6
		THIS^.ipArguments.AddLReal(stCommand.stMoveModuloParameter.fAbsolutePosition);		//7
		THIS^.ipArguments.AddLReal(stCommand.stMoveModuloParameter.fVelocity);				//8
		THIS^.ipArguments.AddLReal(stCommand.stMoveModuloParameter.fAccel);					//9
		THIS^.ipArguments.AddLReal(stCommand.stMoveModuloParameter.fDecel);					//10
		THIS^.ipArguments.AddLReal(stCommand.stMoveModuloParameter.fJerk);					//11
		THIS^.ipArguments.AddLReal(stCommand.stMoveModuloParameter.fGap);					//12
		
	eMoverCommand_eMoveRel:
		THIS^.ipArguments.Clear();													
		THIS^.ipArguments.AddString(stCommand.sText);									//0	
		THIS^.ipArguments.AddString(stCommand.sStation);								//1
		THIS^.ipArguments.AddLReal(stActualMotionParameter.fSetModuloPosition);			//2
		THIS^.ipArguments.AddLReal(stActualMotionParameter.fSetPosition);				//3
		THIS^.ipArguments.AddLReal(stActualMotionParameter.fSetVelo);					//4
		THIS^.ipArguments.AddLReal(stActualMotionParameter.fSetAcc);					//5
		THIS^.ipArguments.AddLReal(stCommand.stMoveRelativeParameter.fDistance);		//6
		THIS^.ipArguments.AddLReal(stCommand.stMoveRelativeParameter.fVelocity);		//7
		THIS^.ipArguments.AddLReal(stCommand.stMoveRelativeParameter.fAccel);			//8
		THIS^.ipArguments.AddLReal(stCommand.stMoveRelativeParameter.fDecel);			//9
		THIS^.ipArguments.AddLReal(stCommand.stMoveRelativeParameter.fJerk);			//10
		THIS^.ipArguments.AddLReal(stCommand.stMoveRelativeParameter.fGap);				//11
			
	eMoverCommand_eGearIn:
		THIS^.ipArguments.Clear();													
		THIS^.ipArguments.AddString(stCommand.sText);									//0	
		THIS^.ipArguments.AddString(stCommand.sStation);								//1
		THIS^.ipArguments.AddLReal(stCommand.stActualMasterParameter.fSetPosition);		//2
		THIS^.ipArguments.AddLReal(stCommand.stActualMasterParameter.fSetVelo);			//3	
		THIS^.ipArguments.AddLReal(stActualMotionParameter.fSetModuloPosition);			//4
		THIS^.ipArguments.AddLReal(stActualMotionParameter.fSetPosition);				//5
		THIS^.ipArguments.AddLReal(stActualMotionParameter.fSetVelo);					//6
		THIS^.ipArguments.AddLReal(stActualMotionParameter.fSetAcc);					//7
		THIS^.ipArguments.AddLReal(stCommand.stGearInParameter.fMasterSyncPosition);	//8
		THIS^.ipArguments.AddLReal(stCommand.stGearInParameter.fMasterStartDistance);	//9
		THIS^.ipArguments.AddLReal(stCommand.stGearInParameter.fSlaveSyncPosition);		//10
		THIS^.ipArguments.AddLReal(stCommand.stGearInParameter.fAbsolutePosition);		//11			
		THIS^.ipArguments.AddLReal(stCommand.stGearInParameter.fAccel);					//12
		THIS^.ipArguments.AddLReal(stCommand.stGearInParameter.fDecel);					//13
		THIS^.ipArguments.AddLReal(stCommand.stGearInParameter.fJerk);					//14
		THIS^.ipArguments.AddLReal(stCommand.stGearInParameter.fGap);					//15
							
	eMoverCommand_eReset:
		THIS^.ipArguments.Clear();
		THIS^.ipArguments.AddString(stCommand.sText);									//0
		THIS^.ipArguments.AddString(stCommand.sStation);								//1
		THIS^.ipArguments.AddLReal(stActualMotionParameter.fSetModuloPosition);			//2	
			
	eMoverCommand_eHaltCa:
		THIS^.ipArguments.Clear();
		THIS^.ipArguments.AddString(stCommand.sText);									//0
		THIS^.ipArguments.AddString(stCommand.sStation);								//1
		THIS^.ipArguments.AddLreal(stActualMotionParameter.fSetModuloPosition);
		THIS^.ipArguments.AddLReal(stCommand.stHaltParameter.fDeceleration);
		THIS^.ipArguments.AddLReal(stCommand.stHaltParameter.fJerk);
		THIS^.ipArguments.AddLReal(stCommand.stHaltParameter.fGap);			
			
	eMoverCommand_eMoveModDone, eMoverCommand_eMoveAbsDone, eMoverCommand_eMoveModQueueing,eMoverCommand_eMoveAbsQueueing :
		THIS^.ipArguments.Clear();
		THIS^.ipArguments.AddString(stCommand.sText);
		THIS^.ipArguments.AddString(stCommand.sStation);			
			
	eMoverCommand_eGearInInSync:
		THIS^.ipArguments.Clear();
		THIS^.ipArguments.AddLReal(stCommand.stActualMasterParameter.fSetPosition);
		THIS^.ipArguments.AddLReal(stCommand.stActualParameter.fSetModuloPosition);
		THIS^.ipArguments.AddString(stCommand.sStation);
	

	eMoverCommand_eGearOutOfSync:
		THIS^.ipArguments.Clear();
		THIS^.ipArguments.AddLreal(stCommand.stActualMasterParameter.fSetPosition);
		THIS^.ipArguments.AddLreal(stCommand.stActualParameter.fSetModuloPosition);
		THIS^.ipArguments.AddString(stCommand.sStation);		
		
	
		eMoverCommand_eHalt:
		THIS^.ipArguments.Clear();
		THIS^.ipArguments.AddString(stCommand.sText);									//0
		THIS^.ipArguments.AddString(stCommand.sStation);								//1
		THIS^.ipArguments.AddLReal(stCommand.stHaltParameter.fDeceleration);
		THIS^.ipArguments.AddLReal(stCommand.stHaltParameter.fJerk);	
		
	*)
END_CASE
THIS^.Send(0);
hresult := THIS^.Release();
END_METHOD

METHOD SetSucceeded : HRESULT
VAR_INPUT
END_VAR
IF NOT THIS^.EqualsToEventEntryEx( stOther := SUCCESS_EVENT) THEN
	THIS^.CreateEx(SUCCESS_EVENT, 0);
END_IF
END_METHOD

END_FUNCTION_BLOCK

// XPlanarStandardFunctions/JoinClosestTrack/FB_JoinClosestTrack
FUNCTION_BLOCK FB_JoinClosestTrack
VAR
	_mover				: I_XPlanarMoverStandard;										// Mover to handle during recovery
	_tracks				: ARRAY[1..Params_XPlanar.maxTrackCount] OF I_TrackStandard;	// Available tracks for recovery

	{attribute 'hide'}
	_velo				: LREAL;
	{attribute 'hide'}
	_acc				: LREAL;
	{attribute 'hide'}
	_dec				: LREAL;
	{attribute 'hide'}
	_jerk				: LREAL;

	{attribute 'hide'}
	_count				: UDINT;														// Qty of tracks in the availability list
	{attribute 'hide'}
	_locked				: BOOL;															// Mover is locked - Cannot recover automatically

	nState				: UDINT;														// State Machine for Execute method
	_distanceToTrack	: ARRAY[1..Params_XPlanar.maxTrackCount] OF ST_TrackDistance;
	_reachPossibility	: ARRAY[1..Params_XPlanar.maxTrackCount] OF ST_TrackReachingTrial;
END_VAR

METHOD AddTrack : BOOL;
VAR_INPUT
	track	: I_TrackStandard;	// Available track for recovery.
END_VAR
IF track = 0 THEN
	// Invalid object itf
	AddTrack := FALSE;
ELSE
	IF _count >= Params_XPlanar.maxTrackCount THEN
		// List already full
		AddTrack := FALSE;
	ELSIF track.P_TrackRef^.MCTOPLC_STD.State = MC_PLANAR_STATE.Invalid THEN
		// NC track not linked
		AddTrack := FALSE;
	ELSE
		// Add Track as last in list
		_tracks[_count + 1] := track;
		_count := _count + 1;
		AddTrack := TRUE;
	END_IF
END_IF
END_METHOD

METHOD AssignMover
VAR_INPUT
	mover			: I_XPlanarMoverStandard;	// Mover to be handled.
	velocity		: LREAL;					// Velocity used during recovery.
	acceleration	: LREAL;					// Acceleration used during recovery.
	deceleration	: LREAL;					// Deceleration used during recovery.
	jerk			: LREAL;					// Jerk used during recovery.
END_VAR
IF mover <> 0 THEN
	_mover := mover;

	_velo := velocity;
	_acc := acceleration;
	_dec := deceleration;
	_jerk := jerk;
END_IF
END_METHOD

METHOD ClearTracks
MEMSET(destAddr:= ADR(_tracks), fillByte:= 0, n:= SIZEOF(_tracks));

_count := 0;
END_METHOD

{attribute 'monitoring' := 'call'}
PROPERTY Locked : BOOL
GET
Locked := _locked;
END_GET
END_PROPERTY

{attribute 'monitoring' := 'call'}
PROPERTY TracksCount : UDINT
GET
TracksCount := _count;
END_GET
END_PROPERTY

METHOD Execute : BOOL
VAR_INPUT
	bReset				: BOOL;		// Reset sequence
END_VAR
VAR_INST
	curPosition			: PositionXYC;
	optionsLeaveTrack	: ST_LeaveTrackOptions	:= (useOrientation:= TRUE);

	optionsMoveC		: ST_MoveCOptions	:= (additionalTurns:= 0, direction:= Tc3_Mc3PlanarMotion.MC_DIRECTION.mcDirectionNonModulo);

	targetPos			: PositionXYC;
	trackIdx			: UDINT;
	targetLocation		: MoverVector;
	xDist				: LREAL;
	yDist				: LREAL;
	optionsMoveToPos	: ST_MoveToPositionOptions	:= (useOrientation:= TRUE);
	insertAtIdx			: UDINT;
	trialIdx			: UDINT;

	joiningBusy			: BOOL;
	moverOnTrack		: OTCID;

	optionsJoinTrack	: ST_JoinTrackOptions	:= (useOrientation:= TRUE);
	joiningErrorInfo	: ST_ErrorDetails;
	moverJoined			: OTCID;

	TON_Timeout			: TON	:= (PT:= T#2S);
	
	nErrorCnt33104		: UINT;
END_VAR
IF bReset THEN
	nErrorCnt33104 := 0;
	_mover := 0;
	nState := 0;
ELSIF nState = 0 THEN
	nState := nState + 1;
END_IF

CASE nState OF
	1:	// Init - Wait for assignments
		_locked := FALSE;
		TON_Timeout(IN:= FALSE);
		IF _mover <> 0 THEN
			IF _count > 0 THEN
				nState := nState + 1;
			END_IF
		END_IF

	2:	// Re-check mover state & reset if errored
		IF _mover.P_State = MC_PLANAR_STATE.Error THEN
			_mover.Reset(slogMessage:= 'Reset error state via FB_Recoverer');
			nState := nState + 1;
		ELSIF _mover.P_State = MC_PLANAR_STATE.Enabled THEN
			nState := nState + 8;
		ELSE
			nState := nState + 1;
		END_IF

	3:	// Resetting mover error (wait for steady state)
		IF _mover.P_State = MC_PLANAR_STATE.Disabled THEN
			nState := nState + 2;
		ELSIF _mover.P_State = MC_PLANAR_STATE.Enabled THEN
			nState := nState + 7;
		END_IF

	5:	// Error Mover locked - Mover is disabled (not in C.A. group anymore)
		_locked := TRUE;


	10:	// Abort pending command
		optionsMoveToPos.useOrientation := TRUE;
		IF _mover.P_Busy THEN
			_mover.Halt(slogMessage:= 'Abort pending cmd');
			nState := nState + 1;
		ELSE
			nState := nState + 2;
		END_IF

	11:
		IF _mover.P_Halt.Done AND NOT _mover.P_Busy THEN
			nState := nState + 1;
		ELSIF _mover.P_Halt.Error THEN
			nState := nState - 9;
		END_IF

	12:	// Set mover to FreeMovement mode
		IF _mover.P_CommandMode = MC_PLANAR_MOVER_COMMAND_MODE.JoiningTrack OR _mover.P_CommandMode = MC_PLANAR_MOVER_COMMAND_MODE.OnTrack OR _mover.P_CommandMode = MC_PLANAR_MOVER_COMMAND_MODE.CRotationOnTrack THEN
			curPosition.SetValuesXYC(x:= _mover.P_SetPosition.x, y:= _mover.P_SetPosition.y, c:= _mover.P_ClosestQuaterAngle);
			_mover.LeaveTrack(slogMessage:= 'Leave cur. track with quadrant align.', position:= curPosition, velocity:= _velo, acceleration:= _acc, deceleration:= _dec, jerk:= _jerk, stOptions:= optionsLeaveTrack);
		ELSIF _mover.P_CommandMode = MC_PLANAR_MOVER_COMMAND_MODE.ExternalSetpointGeneration THEN
			_mover.DisableExternalSetpointGeneration(slogMessage:= 'Stop ext. setpoint gen.');
		END_IF
		nState := nState + 1;

	13:
		IF _mover.P_CommandMode = MC_PLANAR_MOVER_COMMAND_MODE.FreeMovement THEN
			nState := nState + 7;
		ELSIF _mover.P_CommandMode = MC_PLANAR_MOVER_COMMAND_MODE.CRotationFreeMovement THEN
			nState := nState + 1;
		ELSIF _mover.P_LeaveTrack.ErrorID = 33160 AND (_mover.P_CommandMode = MC_PLANAR_MOVER_COMMAND_MODE.OnTrack OR _mover.P_CommandMode = MC_PLANAR_MOVER_COMMAND_MODE.CRotationOnTrack) THEN
			// Track was not standing for Leave command - Retry
			nState := nState - 1;
		END_IF

	14:	// Bring C rotation back to closest quarter turn
		_mover.MoveC(slogMessage:= 'Bring C back to closest quadrant', targetPosition:= _mover.P_ClosestQuaterAngle, velocity:= _velo, acceleration:= _acc, deceleration:= _dec, jerk:= _jerk, stOptions:= optionsMoveC);
		nState := nState + 1;

	15:
		IF _mover.P_MoveC.Done AND _mover.P_CommandMode = MC_PLANAR_MOVER_COMMAND_MODE.FreeMovement THEN
			nState := nState - 2;
		ELSIF _mover.P_MoveC.Error THEN
			nState := nState + 2;
		END_IF

	17:	// Error Mover locked - Cannot rotate C back to closest quadrant
		_locked := TRUE;


	20:	// Determine the joining distance to each available track
		MEMSET(ADR(_distanceToTrack), 0, SIZEOF(_distanceToTrack));
		MEMSET(ADR(_reachPossibility), 0, SIZEOF(_reachPossibility));
		MEMSET(ADR(joiningErrorInfo), 0, SIZEOF(joiningErrorInfo));
		trackIdx := 0;
		nState := nState + 1;

	21:	// Inc track index
		trackIdx := trackIdx + 1;
		IF trackIdx > _count THEN
			nState := nState + 9;
		ELSE
			nState := nState + 1;
		END_IF

	22:	// Fill distance to track characteristics table entry - Check plausability via fake MoveToPosition command (velo = 0)
		_distanceToTrack[trackIdx].Index := trackIdx;
		_distanceToTrack[trackIdx].TrackOID := _tracks[trackIdx].P_OID;
		_distanceToTrack[trackIdx].CurrentLocation := _mover.P_SetPosition;
		curPosition.SetValuesXYC(x:= _distanceToTrack[trackIdx].CurrentLocation.x, y:= _distanceToTrack[trackIdx].CurrentLocation.y, c:= _distanceToTrack[trackIdx].CurrentLocation.c);
		_distanceToTrack[trackIdx].PositionOnTrack := _tracks[trackIdx].GetTrackPositionAt(Position:= curPosition);
		_tracks[trackIdx].GetMoverPositionAt(arcLength:= _distanceToTrack[trackIdx].PositionOnTrack, position:= targetPos);
		_distanceToTrack[trackIdx].TargetLocation.x := targetPos.x;
		_distanceToTrack[trackIdx].TargetLocation.y := targetPos.y;
		_distanceToTrack[trackIdx].TargetLocation.c := _mover.P_ClosestQuaterAngle;
		xDist := ABS(_distanceToTrack[trackIdx].TargetLocation.x - _distanceToTrack[trackIdx].CurrentLocation.x);
		yDist := ABS(_distanceToTrack[trackIdx].TargetLocation.y - _distanceToTrack[trackIdx].CurrentLocation.y);
		_distanceToTrack[trackIdx].Distance := SQRT(EXPT(xDist, 2) + EXPT(yDist, 2));
		targetPos.SetValuesXYC(x:= _distanceToTrack[trackIdx].TargetLocation.x, y:= _distanceToTrack[trackIdx].TargetLocation.y, c:= _distanceToTrack[trackIdx].TargetLocation.c);
		_mover.MoveToPositionExt(slogMessage:= 'Sim. mvt for validity', targetPosition:= targetPos, velocity:= 1E-6, acceleration:= _acc, deceleration:= _dec, jerk:= _jerk, optionsMoveToPos);
		nState := nState + 1;

	23:	// Analyze feedback
		IF _mover.P_MoveToPositionExt.Error THEN
			_distanceToTrack[trackIdx].IsPossibleTrack := FALSE;
			_distanceToTrack[trackIdx].ErrorID := _mover.P_MoveToPositionExt.ErrorID;
			_distanceToTrack[trackIdx].objectInfo.ObjectType := TO_UINT(_mover.P_MoveToPositionExt.stInfo.nObjectType);
			_distanceToTrack[trackIdx].objectInfo.Id := _mover.P_MoveToPositionExt.stInfo.nObjectID;
			nState := nState + 1;
		ELSIF _mover.P_MoveToPositionExt.Active OR _mover.P_MoveToPositionExt.Done THEN
			_distanceToTrack[trackIdx].IsPossibleTrack := TRUE;
			nState := nState + 3;
		END_IF

	24:	// Reset error
		IF _mover.P_State = MC_PLANAR_STATE.Error THEN
			_mover.Reset(slogMessage:= 'Failed - Reset cmd');
			nState := nState + 1;
		ELSIF _mover.P_State = MC_PLANAR_STATE.Enabled THEN
			nState := nState - 3;
		ELSIF _mover.P_State = MC_PLANAR_STATE.Disabled THEN
			nState := nState - 22;
		END_IF

	25:
		IF _mover.P_Reset.Done AND _mover.P_State = MC_PLANAR_STATE.Enabled THEN
			nState := nState - 4;
		ELSIF _mover.P_Reset.Done AND _mover.P_State = MC_PLANAR_STATE.Disabled THEN
			nState := nState - 20;
		END_IF

	26:	// Stopping MoveToPosition trial
		_mover.Halt(slogMessage:= 'Succeed - Abort zero mvt');
		nState := nState + 1;

	27:
		IF _mover.P_Halt.Done AND NOT _mover.P_Busy THEN
			nState := nState + 1;
		END_IF

	28:	// Retain possibility (sort from closest to furthest distance to track)
		insertAtIdx := 1;
		WHILE insertAtIdx <= _count DO
			IF _reachPossibility[insertAtIdx].TrackInfo.TrackOID = 0 OR _reachPossibility[insertAtIdx].TrackInfo.Distance > _distanceToTrack[trackIdx].Distance THEN
				EXIT;
			ELSE
				insertAtIdx := insertAtIdx + 1;
			END_IF
		END_WHILE
		IF insertAtIdx <= _count THEN
			nState := nState + 1;
		END_IF

	29:	// Insert possibility at assigned rank
		FOR trialIdx := _count TO insertAtIdx BY -1 DO
			IF trialIdx = insertAtIdx THEN
				_reachPossibility[trialIdx].TrackInfo := _distanceToTrack[trackIdx];
			ELSIF trialIdx > 1 THEN
				_reachPossibility[trialIdx] := _reachPossibility[trialIdx - 1];
			END_IF
		END_FOR
		nState := nState - 8;


	30:	// Try reaching the closest possible track
		moverOnTrack := 0;
		optionsJoinTrack.useOrientation := optionsMoveToPos.useOrientation;
		trialIdx := 0;
		nState := nState + 1;

	31:
		trialIdx := trialIdx + 1;
		IF trialIdx > _count THEN
			nState := nState + 9;
		ELSE
			nState := nState + 1;
		END_IF

	32:	// Move to track location
		IF NOT _reachPossibility[trialIdx].Busy AND NOT _reachPossibility[trialIdx].Done AND NOT _reachPossibility[trialIdx].Error THEN
			IF _reachPossibility[trialIdx].TrackInfo.TrackOID = 0 THEN
				// Empty possibility - Mark as error for info (process tracking)
				_reachPossibility[trialIdx].Error := TRUE;
				_reachPossibility[trialIdx].ErrorID := 16#FFFFFFFF;
				nState := nState - 1;
			ELSIF _mover.P_CommandMode = MC_PLANAR_MOVER_COMMAND_MODE.FreeMovement THEN
				_reachPossibility[trialIdx].Busy := TRUE;
				targetPos.SetValuesXYC(x:= _reachPossibility[trialIdx].TrackInfo.TargetLocation.x, y:= _reachPossibility[trialIdx].TrackInfo.TargetLocation.y, c:= _reachPossibility[trialIdx].TrackInfo.TargetLocation.c);
				_mover.MoveToPositionExt(slogMessage:= 'Move to track', targetPosition:= targetPos, velocity:= _velo, acceleration:= _acc, deceleration:= _dec, jerk:= _jerk, optionsMoveToPos);
				nState := nState + 1;
			END_IF
		END_IF

	33:	// Moving to track location
		IF _mover.P_MoveToPositionExt.Error THEN
			// Movement failed - Investigate context manually
			_reachPossibility[trialIdx].Busy := FALSE;
			_reachPossibility[trialIdx].Error := TRUE;
			_reachPossibility[trialIdx].ErrorID := _mover.P_MoveToPositionExt.ErrorID;
			_reachPossibility[trialIdx].objectInfo.ObjectType := TO_UINT(_mover.P_MoveToPositionExt.stInfo.nObjectType);
			_reachPossibility[trialIdx].objectInfo.Id := _mover.P_MoveToPositionExt.stInfo.nObjectID;
			moverOnTrack := 0;
			nState := nState - 2;
		ELSIF _mover.P_MoveToPositionExt.Done THEN
			// Success
			_reachPossibility[trialIdx].Busy := FALSE;
			_reachPossibility[trialIdx].Done := TRUE;
			moverOnTrack := _reachPossibility[trialIdx].TrackInfo.TrackOID;
			nState := nState + 7;
		END_IF


	40:	// Try JoinTrack command
		IF moverOnTrack = 0 THEN
			nState := nState + 1;
		ELSE
			TON_Timeout(IN:= TRUE);
			IF (_tracks[_reachPossibility[trialIdx].TrackInfo.Index].P_State = MC_PLANAR_STATE.Enabled AND (_tracks[_reachPossibility[trialIdx].TrackInfo.Index].P_OperationMode = MC_PLANAR_TRACK_OPERATION_MODE.Standing OR _tracks[_reachPossibility[trialIdx].TrackInfo.Index].P_OperationMode = MC_PLANAR_TRACK_OPERATION_MODE.Configuring) AND _mover.P_State = MC_PLANAR_STATE.Enabled) OR TON_Timeout.Q THEN
				TON_Timeout(IN:= FALSE);
				_mover.JoinTrack(slogMessage:= 'Join track', ipTrack:= _tracks[_reachPossibility[trialIdx].TrackInfo.Index], fVelo:= _velo, fAcceleration:= _acc, fJerk:= _jerk, stOptions:= optionsJoinTrack);
				nState := nState + 2;
			END_IF
		END_IF

	41:	// Error Mover locked - No reachable track found
		IF optionsMoveToPos.useOrientation (*EDCA AND _mover.P_ClosestQuaterAngle <> 0*) THEN
			// Twisted mover - Retry without track orientation (but C.A. zone will extend to circle)
			optionsMoveToPos.useOrientation := FALSE;
			nState := 20;
		ELSE
			_locked := TRUE;
		END_IF

	42:
		IF _mover.P_JoinTrack.Error THEN
			// JoinTrack failed - Investigate context manually
			moverJoined := 0;
			joiningErrorInfo.TrackOID := moverOnTrack;
			joiningErrorInfo.ErrorID := _mover.P_JoinTrack.ErrorID;
			joiningErrorInfo.objectInfo.ObjectType := TO_UINT(_mover.P_JoinTrack.stInfo.nObjectType);
			joiningErrorInfo.objectInfo.Id := _mover.P_JoinTrack.stInfo.nObjectID;
			IF optionsJoinTrack.useOrientation AND _mover.P_JoinTrack.ErrorID = 33154 THEN
				// Failed due to twisted mover (C rotation <> track orientation) - Retry without track orientation (but C.A. zone will extend to circle)
				optionsJoinTrack.useOrientation := NOT optionsJoinTrack.useOrientation;
				nState := nState - 2;
			ELSIF NOT optionsJoinTrack.useOrientation AND _mover.P_JoinTrack.ErrorID = 33158 AND _mover.P_ClosestQuaterAngle = 0.0 THEN
				// Failed due to collision avoidance - Retrywith track orientation to reduce C.A. zone (works only if mover C angle is aligned to track)
				optionsJoinTrack.useOrientation := NOT optionsJoinTrack.useOrientation;
				nState := nState - 2;
			ELSIF _mover.P_JoinTrack.ErrorID = 33104 AND nErrorCnt33104 <= 4 THEN
				nErrorCnt33104 := nErrorCnt33104 +1;
				optionsJoinTrack.useOrientation := NOT optionsJoinTrack.useOrientation;
				nState := nState - 2;
			ELSE
				// Failed - Investigate context manually
				nState := nState + 3;
			END_IF
		ELSIF _mover.P_JoinTrack.Done THEN
			// Success
			moverJoined := moverOnTrack;
			nState := nState + 8;
		END_IF

	45:	// Error Mover locked - Cannot join track
		_locked := TRUE;


	50:	// Done
		nState := 255;
END_CASE

Execute := nState = 255;
END_METHOD

END_FUNCTION_BLOCK

// XPlanarStandardFunctions/Mover/I_XPlanarMoverStandard
INTERFACE I_XPlanarMoverStandard EXTENDS __SYSTEM.IQueryInterface

{attribute 'hide'}
PROPERTY P_DcTimeStamp : ULINT
GET
END_GET
END_PROPERTY


METHOD CheckStartConditions : ST_CheckStartConditionFeedback
END_METHOD

METHOD GetCustomTrackID : DINT
VAR_INPUT
END_VAR
END_METHOD

METHOD GetDistanceToTrack : LREAL

VAR_INPUT
	ipTrack	: I_TrackStandard;
END_VAR
END_METHOD

METHOD GetLastKnownCustomTrackID : DINT
VAR_INPUT
END_VAR
END_METHOD

METHOD MoveOnTrack : BOOL
VAR_INPUT
	slogMessage			: STRING;
	ipTrack				: I_TrackStandard;
	trackPosition       : LREAL;
	velocity           	: LREAL;
	acceleration        : LREAL;
	jerk                : LREAL;
	gap					: LREAL;
	direction			: Tc3_Mc3PlanarMotion.MC_DIRECTION;
END_VAR
END_METHOD


{attribute 'obsolete' := 'Obsolete: Please use MoveToPositionExt instead'}
METHOD MoveToPosition  : BOOL
VAR_INPUT
	slogMessage		: STRING;;
	targetPosition	: REFERENCE TO PositionXYC;
	velocity		: LREAL;
	acceleration	: LREAL;
	deceleration	: LREAL;
	jerk			: LREAL;
END_VAR
END_METHOD

METHOD AddToGroup : BOOL
VAR_INPUT
	group : REFERENCE TO MC_PlanarGroup;
END_VAR
END_METHOD

METHOD AdoptTrackOrientation : BOOL
VAR_INPUT
	slogMessage		: STRING;
	velocity		: LREAL;
	acceleration	: LREAL;
	deceleration	: LREAL;
	jerk			: LREAL;
	stOptions 		: REFERENCE TO ST_AdoptTrackOrientationOptions;
END_VAR
END_METHOD

METHOD Disable : BOOL
VAR_INPUT
	slogMessage: STRING;
END_VAR
END_METHOD

METHOD DisableExternalSetpointGeneration : BOOL
VAR_INPUT
	slogMessage : STRING;
END_VAR
END_METHOD

METHOD Enable : BOOL
VAR_INPUT
	slogMessage		: STRING;
END_VAR
END_METHOD

METHOD EnableExternalSetpointGeneration : BOOL
VAR_INPUT
	slogMessage : STRING;
	eSetpointMode : MC_EXTERNAL_SET_POSITION_MODE;
END_VAR
END_METHOD

METHOD GearInPosOnTrack : BOOL
VAR_INPUT
	slogMessage		: STRING;
	master			: OTCID;
	trackTrail		: REFERENCE TO MC_PlanarTrackTrail;
	masterSyncPos	: LREAL;
	slaveSyncPos	: LREAL;
	syncTrack		: I_TrackStandard;
	velocity		: LREAL;
	acceleration	: LREAL;
	deceleration	: LREAL;
	jerk			: LREAL;
	stOptions 		: REFERENCE TO ST_GearInPosOnTrackOptions;
END_VAR
END_METHOD

METHOD GetCommandLog : ST_MoverCommandLog
VAR_INPUT
	nNum	: UINT;
END_VAR
END_METHOD

METHOD GetPositionOnCurrentPart : BOOL
VAR_IN_OUT
	position : PositionXYC;
END_VAR
END_METHOD

METHOD Halt : BOOL
VAR_INPUT
	slogMessage		: STRING;
END_VAR
END_METHOD

METHOD JoinTrack : BOOL
VAR_INPUT
	slogMessage		: STRING;
	ipTrack 		: I_TrackStandard;
	fVelo			: LREAL;
	fAcceleration	: LREAL;
	fJerk			: LREAL;
	stOptions		: REFERENCE TO ST_JoinTrackOptions;
END_VAR
END_METHOD

METHOD LeaveTrack : BOOL
VAR_INPUT
	slogMessage		: STRING;
	position 		: REFERENCE TO PositionXYC;
	velocity 		: LREAL;
	acceleration	: LREAL;
	deceleration	: LREAL;
	jerk			: LREAL;
	stOptions		: REFERENCE TO ST_LeaveTrackOptions;
END_VAR
END_METHOD

METHOD LeaveTrackInPosition : BOOL
VAR_INPUT
	slogMessage		: STRING;
	bUseOrientation	: BOOL;
END_VAR
END_METHOD

METHOD MoveA : BOOL
VAR_INPUT
	slogMessage		: STRING;
	targetPosition	: LREAL;
	velocity		: LREAL;
	acceleration	: LREAL;
	deceleration	: LREAL;
	jerk			: LREAL;
END_VAR
END_METHOD

METHOD MoveB : BOOL
VAR_INPUT
	slogMessage		: STRING;
	targetPosition	: LREAL;
	velocity		: LREAL;
	acceleration	: LREAL;
	deceleration	: LREAL;
	jerk			: LREAL;
END_VAR
END_METHOD

METHOD MoveC : BOOL
VAR_INPUT
	slogMessage		: STRING;
	targetPosition	: LREAL;
	velocity		: LREAL;
	acceleration	: LREAL;
	deceleration	: LREAL;
	jerk			: LREAL;
	stOptions		: REFERENCE TO ST_MoveCOptions;
END_VAR
END_METHOD

METHOD MoveOnTrackExt : BOOL
VAR_INPUT
	sLogMessage				: STRING;
	ipTrack					: I_TrackStandard;
	trackPosition       	: LREAL;
	velocity           		: LREAL;
	acceleration        	: LREAL;
	jerk                	: LREAL;
	stMoveOnTrackOptions	: ST_MoveOnTrackOptions;
END_VAR
END_METHOD

METHOD MoveToPositionExt  : BOOL
VAR_INPUT
	slogMessage					: STRING;
	targetPosition				: REFERENCE TO PositionXYC;
	velocity					: LREAL;
	acceleration				: LREAL;
	deceleration				: LREAL;
	jerk						: LREAL;
	stMoveToPositionOptions		: ST_MoveToPositionOptions;
END_VAR
END_METHOD

{attribute 'hide'}
{attribute 'obsolete' := 'Obsolete: Please use MoveToPositionExt instead'}
METHOD MoveToPositionXYC  : BOOL
VAR_INPUT
	slogMessage		: STRING;
	targetPosition	: REFERENCE TO PositionXYC;
	velocity		: LREAL;
	acceleration	: LREAL;
	deceleration	: LREAL;
	jerk			: LREAL;
END_VAR
END_METHOD

METHOD MoveZ : BOOL
VAR_INPUT
	slogMessage		: STRING;
	targetPosition	: LREAL;
	velocity		: LREAL;
	acceleration	: LREAL;
	deceleration	: LREAL;
	jerk			: LREAL;
END_VAR
END_METHOD

METHOD RemoveFromGroup : BOOL
VAR_INPUT
END_VAR
END_METHOD

METHOD Reset : BOOL
VAR_INPUT
	slogMessage 	: STRING;;
END_VAR
END_METHOD

METHOD SetExternalSetpointValues : BOOL
VAR_INPUT
	position 		: MoverVector;
	velocity 		: MoverVector;
	acceleration 	: MoverVector;
END_VAR
END_METHOD

METHOD SetMoverPosition : BOOL

VAR_INPUT
	slogMessage		: STRING;
	position		: REFERENCE TO PositionXYC;
END_VAR
END_METHOD

PROPERTY P_AtRotationPoint : BOOL
GET
END_GET
END_PROPERTY

PROPERTY P_ClosestQuaterAngle : LREAL
GET
END_GET
END_PROPERTY

PROPERTY P_CRotationRestrictions : BOOL
GET
END_GET
END_PROPERTY

PROPERTY P_CustomTrackIdTable : ARRAY [1..Params_XPlanar.maxTrackCount] OF ST_CutomTrackID;
SET
END_SET
END_PROPERTY

PROPERTY P_HaltDynamics : ST_HaltDynamics
GET
END_GET
SET
END_SET
END_PROPERTY

PROPERTY P_IsMovingXY : BOOL
GET
END_GET
END_PROPERTY

PROPERTY P_IsPresent : BOOL
GET
END_GET
END_PROPERTY

PROPERTY P_IsQueuing : BOOL
GET
END_GET
END_PROPERTY

PROPERTY P_IsSetpointGeneratorActive : BOOL
GET
END_GET
END_PROPERTY

PROPERTY P_LastKnownTrackOID : OTCID
GET
END_GET
END_PROPERTY

PROPERTY P_RotationAngleModulo : LREAL
GET
END_GET
END_PROPERTY

PROPERTY P_SavedMoveOnTrackParameter : REFERENCE TO ST_MoveOnTrackParameters
GET
END_GET
END_PROPERTY


PROPERTY P_ZeroVelocityThreshold : LREAL
GET
END_GET
SET
END_SET
END_PROPERTY

PROPERTY P_AddToGroup : REFERENCE TO ST_CommandReturn
GET
END_GET
END_PROPERTY

PROPERTY P_AdoptTrackOrientation : REFERENCE TO ST_CommandReturn
GET
END_GET
END_PROPERTY

PROPERTY P_Disable : REFERENCE to ST_CommandReturn
GET
END_GET
END_PROPERTY

PROPERTY P_DisableExternalSetpointGeneration : REFERENCE to ST_CommandReturn
GET
END_GET
END_PROPERTY

PROPERTY P_Enable : REFERENCE to ST_CommandReturn
GET
END_GET
END_PROPERTY

PROPERTY P_EnableExternalSetpointGeneration : REFERENCE to ST_CommandReturn
GET
END_GET
END_PROPERTY

PROPERTY P_GearInPosOnTrack : REFERENCE TO ST_CommandReturnGearInPosOnTrack
GET
END_GET
END_PROPERTY

PROPERTY P_GearInPosOnTrackMasterMover : REFERENCE TO ST_CommandReturnGearInPosOnTrackWithMasterMover
GET
END_GET
END_PROPERTY

PROPERTY P_Halt : REFERENCE to ST_CommandReturn
GET
END_GET
END_PROPERTY

PROPERTY P_JoinTrack : REFERENCE to ST_CommandReturn
GET
END_GET
END_PROPERTY

PROPERTY P_LeaveTrack : REFERENCE to ST_CommandReturn
GET
END_GET
END_PROPERTY

PROPERTY P_LeaveTrackInPosition : REFERENCE to ST_CommandReturn
GET
END_GET
END_PROPERTY

PROPERTY P_MoveA : REFERENCE to ST_CommandReturn
GET
END_GET
END_PROPERTY

PROPERTY P_MoveB : REFERENCE to ST_CommandReturn
GET
END_GET
END_PROPERTY

PROPERTY P_MoveC : REFERENCE TO ST_CommandReturn
GET
END_GET
END_PROPERTY

PROPERTY P_MoveOnTrack : REFERENCE to ST_CommandReturn
GET
END_GET
END_PROPERTY

PROPERTY P_MoveOnTrackExt : REFERENCE to ST_CommandReturn
GET
END_GET
END_PROPERTY

{attribute 'obsolete' := 'Obsolete: Please use P_MoveToPositionExt instead'}
PROPERTY P_MoveToPosition : REFERENCE to ST_CommandReturn
GET
END_GET
END_PROPERTY


PROPERTY P_MoveToPositionExt : REFERENCE to ST_CommandReturn
GET
END_GET
END_PROPERTY

{attribute 'hide'}
{attribute 'obsolete' := 'Obsolete: Please use P_MoveToPositionExt instead'}
PROPERTY P_MoveToPositionXYC : REFERENCE to ST_CommandReturn
GET
END_GET
END_PROPERTY

PROPERTY P_MoveZ : REFERENCE to ST_CommandReturn
GET
END_GET
END_PROPERTY

PROPERTY P_RemoveFromGroup : REFERENCE TO ST_CommandReturn
GET
END_GET
END_PROPERTY

PROPERTY P_Reset : REFERENCE to ST_CommandReturn
GET
END_GET
END_PROPERTY


PROPERTY P_SetMoverPosition : REFERENCE to ST_CommandReturn
GET
END_GET
END_PROPERTY

PROPERTY P_ActPosition : Reference To MoverVector
GET
END_GET
END_PROPERTY

PROPERTY P_ActVelocity : REFERENCE TO MoverVector
GET
END_GET
END_PROPERTY

PROPERTY P_Busy : BOOL
GET
END_GET
END_PROPERTY

PROPERTY P_CommandMode : MC_PLANAR_MOVER_COMMAND_MODE
GET
END_GET
END_PROPERTY

PROPERTY P_Error : Bool
GET
END_GET
END_PROPERTY

PROPERTY P_ErrorCode : DINT
GET
END_GET
END_PROPERTY

PROPERTY P_ErrorID : UDINT
GET
END_GET
END_PROPERTY

PROPERTY P_Id : UINT
GET
END_GET
SET
END_SET
END_PROPERTY

PROPERTY P_InGroup : BOOL
GET
END_GET
END_PROPERTY

PROPERTY P_MoverOid : OTCID
GET
END_GET
END_PROPERTY

{attribute 'hide'}
PROPERTY P_MoverRef : POINTER TO MC_PlanarMover
GET
END_GET
END_PROPERTY

PROPERTY P_PhysicalAreaID : UDINT
GET
END_GET
END_PROPERTY

PROPERTY P_SetAcceleration : REFERENCE TO MoverVector
GET
END_GET
END_PROPERTY

PROPERTY P_SetOnTrack : Reference To CDT_MCTOPLC_PLANAR_MOVER_TRACK
GET
END_GET
END_PROPERTY

PROPERTY P_SetPosition : REFERENCE TO MoverVector
GET
END_GET
END_PROPERTY

PROPERTY P_SetVelocity : REFERENCE TO MoverVector
GET
END_GET
END_PROPERTY

PROPERTY P_State : MC_PLANAR_STATE
GET
END_GET
END_PROPERTY

PROPERTY P_TrackId : UDINT
GET
END_GET
END_PROPERTY

METHOD Cycle : BOOL
VAR_INPUT
END_VAR
END_METHOD

END_INTERFACE

// XPlanarStandardFunctions/Track/I_TrackStandard
INTERFACE I_TrackStandard EXTENDS __SYSTEM.IQueryInterface

PROPERTY P_AddToGroup : REFERENCE TO ST_CommandReturn
GET
END_GET
END_PROPERTY

PROPERTY P_AppendCircle : REFERENCE TO ST_CommandReturn
GET
END_GET
END_PROPERTY

PROPERTY P_AppendLine : REFERENCE TO ST_CommandReturn
GET
END_GET
END_PROPERTY

PROPERTY P_AppendPoint : REFERENCE TO ST_CommandReturn
GET
END_GET
END_PROPERTY

PROPERTY P_BuildTrack : REFERENCE TO ST_CommandReturn
GET
END_GET
END_PROPERTY

PROPERTY P_BuildTrackAdvanced : REFERENCE TO ST_CommandReturn
GET
END_GET
END_PROPERTY

PROPERTY P_BuildTrackAdvanced_Check : int
GET
END_GET
END_PROPERTY

PROPERTY P_BuildTrackAdvancedInfoText : STRING
GET
END_GET
END_PROPERTY

PROPERTY P_BuildTrackExt : REFERENCE TO ST_CommandReturn
GET
END_GET
END_PROPERTY

PROPERTY P_Clear : REFERENCE TO ST_CommandReturn
GET
END_GET
END_PROPERTY

PROPERTY P_CloseLoop : REFERENCE TO ST_CommandReturn
GET
END_GET
END_PROPERTY

PROPERTY P_Disable : REFERENCE TO ST_CommandReturn
GET
END_GET
END_PROPERTY

PROPERTY P_Enable : REFERENCE TO ST_CommandReturn
GET
END_GET
END_PROPERTY

PROPERTY P_EndAtTrack : REFERENCE TO ST_CommandReturn
GET
END_GET
END_PROPERTY

PROPERTY P_RemoveFromGroup : REFERENCE TO ST_CommandReturn
GET
END_GET
END_PROPERTY

PROPERTY P_Reset : REFERENCE TO ST_CommandReturn
GET
END_GET
END_PROPERTY

PROPERTY P_StartFromTrack : REFERENCE TO ST_CommandReturn
GET
END_GET
END_PROPERTY

METHOD AddToGroup : BOOL
VAR_INPUT
	group : REFERENCE TO MC_PlanarGroup;
END_VAR
END_METHOD

METHOD AppendCircle : BOOL
VAR_INPUT
	startPosition	: REFERENCE TO PositionXYC;
	centerPosition	: REFERENCE TO PositionXY;
	endPosition 	: REFERENCE TO PositionXYC;
	clockwise		: REFERENCE TO BOOL;
END_VAR
END_METHOD

METHOD AppendLine : BOOL
VAR_INPUT
	startPosition	: REFERENCE TO PositionXYC;
	endPosition 	: REFERENCE TO PositionXYC;
END_VAR
END_METHOD

METHOD AppendPoint : BOOL
VAR_INPUT
	position	: REFERENCE TO PositionXYC;
END_VAR
END_METHOD

{attribute 'hide'}
METHOD BuildTrack : BOOL
VAR_INPUT
	TrackTable			: ARRAY [1..maxNumTrackPoints,1..3] OF LREAL;
	ipStartFromTrack	: I_TrackStandard;		
	ipEndAtTrack 		: I_TrackStandard;
	bCloseLoop			: BOOL;
END_VAR
END_METHOD

METHOD BuildTrackAdvanced : BOOL
VAR_INPUT
	TrackTable			: REFERENCE TO FB_TrackTableAdvanced;
END_VAR
END_METHOD

METHOD BuildTrackExt : BOOL
VAR_INPUT
	TrackTable			: REFERENCE TO FB_TrackTable;
END_VAR
END_METHOD

METHOD Clear : BOOL
VAR_INPUT
END_VAR
END_METHOD

METHOD CloseLoop : BOOL
VAR_INPUT
END_VAR
END_METHOD

METHOD Cycle : BOOL
VAR_INPUT
END_VAR
END_METHOD

METHOD Disable : BOOL
VAR_INPUT
END_VAR
END_METHOD

METHOD Enable : BOOL
VAR_INPUT
END_VAR
END_METHOD

METHOD GetCommandLog : ST_TrackCommandLog
VAR_INPUT
	nNum	: UINT;
END_VAR
END_METHOD

METHOD GetLength : LREAL
VAR_INPUT
END_VAR
END_METHOD

METHOD GetMoverPositionAt : BOOL

VAR_INPUT
	(* Arc length value where the position is evaluated. *)
	arcLength : LREAL;
END_VAR
VAR_IN_OUT
	(* The position at the specified arc parameter. *)
	position : PositionXYC;
END_VAR
END_METHOD

METHOD GetTrackPositionAt : LREAL
VAR_INPUT
	Position : REFERENCE TO PositionXYC;
END_VAR
END_METHOD

METHOD GetTrackPositionAt_XY : LREAL
VAR_INPUT
	x	: LREAL;
	y	: LREAL;
END_VAR
END_METHOD

PROPERTY P_GroupOID : UDINT
GET
END_GET
END_PROPERTY

PROPERTY P_Info : PlanarObjectInfo
GET
END_GET
END_PROPERTY

PROPERTY P_MoverCountOnTrack : UDINT
GET
END_GET
END_PROPERTY

PROPERTY P_MovingMoverCount : UDINT
GET
END_GET
END_PROPERTY

PROPERTY P_OID : UDINT
GET
END_GET
END_PROPERTY

PROPERTY P_OperationMode : MC_PLANAR_TRACK_OPERATION_MODE
GET
END_GET
END_PROPERTY

PROPERTY P_State : MC_PLANAR_STATE
GET
END_GET
END_PROPERTY

PROPERTY P_TrackRef : POINTER TO MC_PlanarTrack
GET
END_GET
END_PROPERTY

PROPERTY ref : PVOID
GET
END_GET
END_PROPERTY

METHOD RemoveFromGroup : BOOL
VAR_INPUT
END_VAR
END_METHOD

METHOD Reset : BOOL
VAR_INPUT
END_VAR
END_METHOD

END_INTERFACE

// XPlanarStandardFunctions/Track/FB_TrackTableAdvanced
FUNCTION_BLOCK FB_TrackTableAdvanced


VAR
	
	TrackTable				: ARRAY[1..maxNumTrackPoints] OF ST_TrackTable;
	nTrackTableIndex		: UINT;
	
	sInfoText				: STRING;
	idx						: UINT;
	nStateCheckTabel		: UINT;
	nIndex					: UINT;
	bTrackTablePlausible	: BOOL;
	nTableImplausibleIndex	: UINT;
	
	stTrackBuildParameter	: ST_TrackBuildParameter;
	

	bStartingTrackFailed	: BOOL;
	bEndingTrackFailed		: BOOL;	
	
	bCloseTheLoop			: BOOL;

END_VAR

METHOD AddPoint : INT
VAR_INPUT
	
	ePointType		: E_PointType;
	eOption			: E_PointOption;
	Position_X		: LREAL;
	Position_Y		: LREAL;
	Orientation_C	: LREAL;
	ReferenceSystem : OTCID := 0;

END_VAR


	nTrackTableIndex := nTrackTableIndex +1;

	IF nTrackTableIndex <= maxNumTrackPoints THEN

		TrackTable[nTrackTableIndex].ePointType	    	 := ePointType;
		TrackTable[nTrackTableIndex].eOption		     := eOption;
		TrackTable[nTrackTableIndex].fPointPosition_X    := Position_X;	 
		TrackTable[nTrackTableIndex].fPointPosition_Y    := Position_Y;
		TrackTable[nTrackTableIndex].fPointOrientation_C := Orientation_C;
		TrackTable[nTrackTableIndex].ReferenceSystem     := ReferenceSystem;
		
		sInfoText := 'Track point added sucessfully';
		AddPoint := 1;
	
	ELSE
		sInfoText := 'Error - TrackTable overflow';
		AddPoint := -1;		
	END_IF
END_METHOD

METHOD CheckPoint : ST_TrackPoint
VAR_INPUT
	
	nTackPointIndex	: INT;

END_VAR
	


	IF nTrackTableIndex <= nTrackTableIndex THEN
		CheckPoint.ePointType 		:= TrackTable[nTackPointIndex].ePointType;
		CheckPoint.eOption 			:= TrackTable[nTackPointIndex].eOption;
		CheckPoint.Position_X 		:= TrackTable[nTackPointIndex].fPointPosition_X;
		CheckPoint.Position_Y 		:= TrackTable[nTackPointIndex].fPointPosition_Y;
		CheckPoint.Orientation_C 	:= TrackTable[nTackPointIndex].fPointOrientation_C;
	ELSE
		CheckPoint.ePointType 		:= E_PointType.none;
		CheckPoint.eOption 			:= E_PointOption.none;
		CheckPoint.Position_X 		:= 0.0;
		CheckPoint.Position_Y 		:= 0.0;
		CheckPoint.Orientation_C 	:= 0.0;
	END_IF
END_METHOD

METHOD CheckTrackTable : DINT
VAR_INPUT
END_VAR

	

	CASE nStateCheckTabel OF
		
	0:	
		                nIndex := 1;
		  bTrackTablePlausible := TRUE;
		nTableImplausibleIndex := 0;
				     sInfoText := 'Checking TrackTable';
			   CheckTrackTable := 0;
		      nStateCheckTabel := 90;
	
		
	90:	
		IF nIndex <= maxNumTrackPoints THEN
			nStateCheckTabel := 100;
		ELSE
			nStateCheckTabel := 200;
		END_IF		
			
			
	100:	
		IF TrackTable[nIndex].ePointType = E_PointType.Point THEN
			nStateCheckTabel := 110;
		ELSIF TrackTable[nIndex].ePointType = E_PointType.Line_Start THEN
			nStateCheckTabel := 120;
		ELSIF TrackTable[nIndex].ePointType = E_PointType.Circle_Start THEN
			nStateCheckTabel := 130;
		ELSIF TrackTable[nIndex].ePointType = E_PointType.none THEN
			nStateCheckTabel := 200;
		END_IF
		
		
	110:  // Checking Point	
		IF nIndex+1 <= maxNumTrackPoints THEN 
			nStateCheckTabel := nStateCheckTabel + 5;
		ELSE
			nStateCheckTabel := 200;
		END_IF	
	
	115:
		IF  TrackTable[nIndex +1].ePointType <> E_PointType.Line_End 
		AND TrackTable[nIndex +1].ePointType <> E_PointType.Circle_Center	
		AND TrackTable[nIndex +1].ePointType <> E_PointType.Circle_End
		THEN
		    nIndex := nIndex +1;
			nStateCheckTabel := 90;
		ELSE
			  bTrackTablePlausible := FALSE;
		    nTableImplausibleIndex := nIndex+1;	
				  nStateCheckTabel := 200;		
		END_IF
				
		
	120:  // Checking Line 
		IF nIndex+1 <= maxNumTrackPoints THEN 
			nStateCheckTabel := nStateCheckTabel + 5;
		ELSE
			  bTrackTablePlausible := FALSE;
			nTableImplausibleIndex := nIndex;			
			      nStateCheckTabel := 200;
		END_IF			
	
	125:
		IF TrackTable[nIndex +1].ePointType = E_PointType.Line_End THEN
			nIndex := nIndex +2;
			nStateCheckTabel := 90;	
		ELSE
			  bTrackTablePlausible := FALSE;
		    nTableImplausibleIndex := nIndex+1;
			      nStateCheckTabel := 200;
		END_IF
		
		
	130:  // Checking Circle
		IF nIndex+2 <= maxNumTrackPoints THEN 
			nStateCheckTabel := nStateCheckTabel + 5;
		ELSE
			  bTrackTablePlausible := FALSE;
			nTableImplausibleIndex := nIndex;			
			      nStateCheckTabel := 200;
		END_IF		
	

	135:
		IF  TrackTable[nIndex +1].ePointType = E_PointType.Circle_Center
		AND TrackTable[nIndex +2].ePointType = E_PointType.Circle_End
		THEN
			nIndex := nIndex +3;
			nStateCheckTabel := 90;	
		ELSE
		
			IF TrackTable[nIndex +1].ePointType <> E_PointType.Circle_Center THEN
				nTableImplausibleIndex := nIndex+1;
			ELSE
				nTableImplausibleIndex := nIndex+2;	
			END_IF
			
			bTrackTablePlausible := FALSE;
			    nStateCheckTabel := 200;
		END_IF
		
		
	200: // Check finished
		IF bStartingTrackFailed THEN
			CheckTrackTable := -1;
		 	      sInfoText := 'Start from track implausible!';	
		ELSIF bEndingTrackFailed THEN
			CheckTrackTable := -1;
		 	      sInfoText := 'End at track implausible!';	
		ELSIF bTrackTablePlausible THEN
			CheckTrackTable := 1;
		 	      sInfoText := 'TrackTable check successful';
		ELSE
			CheckTrackTable := -UINT_TO_DINT(nTableImplausibleIndex);
			      sInfoText := CONCAT('TrackTable check failed at track point: ', UINT_TO_STRING(nTableImplausibleIndex));
		END_IF

		nStateCheckTabel := 0;
		
	END_CASE
END_METHOD

METHOD ClearTrackTable : BOOL
VAR_INPUT
END_VAR


	bStartingTrackFailed := FALSE;
	bEndingTrackFailed	 := FALSE;
	
	
	nTrackTableIndex := 0;
	MEMSET(ADR(TrackTable),0,SIZEOF(TrackTable));
	MEMSET(ADR(stTrackBuildParameter),0,SIZEOF(stTrackBuildParameter));
	
	
	sInfoText := 'TrackTable cleared';
	
	ClearTrackTable := TRUE;
END_METHOD

PROPERTY P_BuildlParameter : ST_TrackBuildParameter
GET
	P_BuildlParameter := stTrackBuildParameter;
END_GET
END_PROPERTY

PROPERTY P_CloseTheLoop : BOOL
GET
P_CloseTheLoop := bCloseTheLoop;
END_GET
SET
bCloseTheLoop := P_CloseTheLoop;

IF bCloseTheLoop THEN
	sInfoText := 'Set CloseTheLoop';
ELSE
	sInfoText := 'Cleared CloseTheLoop';
END_IF
END_SET
END_PROPERTY

PROPERTY P_EndAtTrack : I_TrackStandard
GET
	P_EndAtTrack := stTrackBuildParameter.EndAtTrack;
END_GET
SET
IF P_EndAtTrack <> 0 THEN
	IF P_EndAtTrack.ref <> 0 THEN
	      stTrackBuildParameter.EndAtTrack := P_EndAtTrack;
		  
		  bEndingTrackFailed := FALSE;
		           sInfoText := 'Added ending track successfully';
	ELSE
		bEndingTrackFailed := TRUE;
		sInfoText := 'Adding failed, object reference is null!';
	END_IF
ELSE
	bEndingTrackFailed := TRUE;
	sInfoText := 'Adding failed, object is null!';
END_IF
END_SET
END_PROPERTY

PROPERTY P_EndAtTrackOptions : ST_EndAtTrackAdvancedOptions
GET
P_EndAtTrackOptions := stTrackBuildParameter.endOptions;
END_GET
SET
stTrackBuildParameter.endOptions := P_EndAtTrackOptions;
END_SET
END_PROPERTY

PROPERTY P_InfoText : STRING
GET


	P_InfoText := sInfoText;
END_GET
END_PROPERTY

PROPERTY P_NumberOfPointsInTable : UINT
GET
	

	P_NumberOfPointsInTable := nTrackTableIndex;
END_GET
END_PROPERTY

PROPERTY P_StartFromTrack : I_TrackStandard
GET
	P_StartFromTrack := stTrackBuildParameter.StartFromTrack;
END_GET
SET
IF P_StartFromTrack <> 0 THEN
	IF P_StartFromTrack.ref <> 0 THEN
		stTrackBuildParameter.StartFromTrack := P_StartFromTrack;
		
		bStartingTrackFailed := FALSE;
		           sInfoText := 'Added starting track successfully';
	ELSE
		bStartingTrackFailed := TRUE;
		sInfoText := 'Adding failed, object reference is null!';
	END_IF
ELSE
	bStartingTrackFailed := TRUE;
	sInfoText := 'Adding failed, object is null!';
END_IF
END_SET
END_PROPERTY

PROPERTY P_StartFromTrackOptions : ST_StartFromTrackAdvancedOptions
GET
P_StartFromTrackOptions := stTrackBuildParameter.startOptions;
END_GET
SET
stTrackBuildParameter.startOptions := P_StartFromTrackOptions;
END_SET
END_PROPERTY

PROPERTY P_Table : REFERENCE TO ARRAY[1..maxNumTrackPoints] OF ST_TrackTable
GET
P_Table REF= TrackTable;
END_GET
END_PROPERTY

PROPERTY P_TrackCheckImplausibleTableIndex : UINT
GET
P_TrackCheckImplausibleTableIndex := nTableImplausibleIndex;
END_GET
END_PROPERTY

PROPERTY P_TrackTableCheckResult : BOOL
GET
P_TrackTableCheckResult := bTrackTablePlausible;
END_GET
END_PROPERTY

END_FUNCTION_BLOCK

// XPlanarStandardFunctions/Track/FB_TrackTable
FUNCTION_BLOCK FB_TrackTable


VAR
	
	TrackTable				: ARRAY[1..maxNumTrackPoints] OF ST_TrackTable;
	nTrackTableIndex		: UINT;
	sInfoText				: STRING;
	bStartingTrackFailed	: BOOL;
	bEndingTrackFailed		: BOOL;	
	bTrackTablePlausible	: BOOL;
	nTableImplausibleIndex	: UINT;	

	{attribute 'hide'}
	idx						: UINT;
	{attribute 'hide'}
	nStateCheckTabel		: UINT;
	{attribute 'hide'}
	nIndex					: UINT;	
	{attribute 'hide'}
	stTrackBuildParameter	: ST_TrackBuildParameter;
	{attribute 'hide'}
	bCloseTheLoop			: BOOL;

END_VAR

METHOD AddPoint : INT
VAR_INPUT
	
	ePointType		: E_PointType;
	eOption			: E_PointOption;
	Position_X		: LREAL;
	Position_Y		: LREAL;
	Orientation_C	: LREAL;

END_VAR


	nTrackTableIndex := nTrackTableIndex +1;

	IF nTrackTableIndex <= maxNumTrackPoints THEN

		TrackTable[nTrackTableIndex].ePointType	    	 := ePointType;
		TrackTable[nTrackTableIndex].eOption		     := eOption;
		TrackTable[nTrackTableIndex].fPointPosition_X    := Position_X;	 
		TrackTable[nTrackTableIndex].fPointPosition_Y    := Position_Y;
		TrackTable[nTrackTableIndex].fPointOrientation_C := Orientation_C;
		
		sInfoText := 'Track point added sucessfully';
		AddPoint := 1;
	
	ELSE
		sInfoText := 'Error - TrackTable overflow';
		AddPoint := -1;		
	END_IF
END_METHOD

METHOD CheckTrackTable : DINT
VAR_INPUT
END_VAR

	

	CASE nStateCheckTabel OF
		
	0:	
		                nIndex := 1;
		  bTrackTablePlausible := TRUE;
		nTableImplausibleIndex := 0;
				     sInfoText := 'Checking TrackTable';
			   CheckTrackTable := 0;
		      nStateCheckTabel := 90;
	
		
	90:	
		IF nIndex <= maxNumTrackPoints THEN
			nStateCheckTabel := 100;
		ELSE
			nStateCheckTabel := 200;
		END_IF		
			
			
	100:	
		IF TrackTable[nIndex].ePointType = E_PointType.Point THEN
			nStateCheckTabel := 110;
		ELSIF TrackTable[nIndex].ePointType = E_PointType.Line_Start THEN
			nStateCheckTabel := 120;
		ELSIF TrackTable[nIndex].ePointType = E_PointType.Circle_Start THEN
			nStateCheckTabel := 130;
		ELSIF TrackTable[nIndex].ePointType = E_PointType.none THEN
			nStateCheckTabel := 200;
		END_IF
		
		
	110:  // Checking Point	
		IF nIndex+1 <= maxNumTrackPoints THEN 
			nStateCheckTabel := nStateCheckTabel + 5;
		ELSE
			nStateCheckTabel := 200;
		END_IF	
	
	115:
		IF  TrackTable[nIndex +1].ePointType <> E_PointType.Line_End 
		AND TrackTable[nIndex +1].ePointType <> E_PointType.Circle_Center	
		AND TrackTable[nIndex +1].ePointType <> E_PointType.Circle_End
		THEN
		    nIndex := nIndex +1;
			nStateCheckTabel := 90;
		ELSE
			  bTrackTablePlausible := FALSE;
		    nTableImplausibleIndex := nIndex+1;	
				  nStateCheckTabel := 200;		
		END_IF
				
		
	120:  // Checking Line 
		IF nIndex+1 <= maxNumTrackPoints THEN 
			nStateCheckTabel := nStateCheckTabel + 5;
		ELSE
			  bTrackTablePlausible := FALSE;
			nTableImplausibleIndex := nIndex;			
			      nStateCheckTabel := 200;
		END_IF			
	
	125:
		IF TrackTable[nIndex +1].ePointType = E_PointType.Line_End THEN
			nIndex := nIndex +2;
			nStateCheckTabel := 90;	
		ELSE
			  bTrackTablePlausible := FALSE;
		    nTableImplausibleIndex := nIndex+1;
			      nStateCheckTabel := 200;
		END_IF
		
		
	130:  // Checking Circle
		IF nIndex+2 <= maxNumTrackPoints THEN 
			nStateCheckTabel := nStateCheckTabel + 5;
		ELSE
			  bTrackTablePlausible := FALSE;
			nTableImplausibleIndex := nIndex;			
			      nStateCheckTabel := 200;
		END_IF		
	

	135:
		IF  TrackTable[nIndex +1].ePointType = E_PointType.Circle_Center
		AND TrackTable[nIndex +2].ePointType = E_PointType.Circle_End
		THEN
			//nIndex := nIndex +3;
			nStateCheckTabel := 140;	
		ELSE
		
			IF TrackTable[nIndex +1].ePointType <> E_PointType.Circle_Center THEN
				nTableImplausibleIndex := nIndex+1;
			ELSE
				nTableImplausibleIndex := nIndex+2;	
			END_IF
			
			bTrackTablePlausible := FALSE;
			    nStateCheckTabel := 200;
		END_IF
		
		
	140:
		IF  TrackTable[nIndex].eOption = E_PointOption.Circle_Clockwise THEN
			IF  TrackTable[nIndex].eOption = E_PointOption.Circle_Clockwise
			AND TrackTable[nIndex+1].eOption = E_PointOption.Circle_Clockwise
			AND TrackTable[nIndex+2].eOption = E_PointOption.Circle_Clockwise
			THEN
				nStateCheckTabel := 145;
			END_IF
		ELSE
			IF  TrackTable[nIndex].eOption = E_PointOption.Circle_CounterClockwise
			AND TrackTable[nIndex+1].eOption = E_PointOption.Circle_CounterClockwise
			AND TrackTable[nIndex+2].eOption = E_PointOption.Circle_CounterClockwise
			THEN
				nStateCheckTabel := 145;
			ELSE
				  bTrackTablePlausible := FALSE;
				nTableImplausibleIndex := nIndex;			
					  nStateCheckTabel := 200;
			END_IF	
		END_IF


	145:
		nIndex := nIndex +3;
		nStateCheckTabel := 90;
		
			
						
		
		
	200: // Check finished
		IF bStartingTrackFailed THEN
			CheckTrackTable := -1;
		 	      sInfoText := 'Start from track implausible!';	
		ELSIF bEndingTrackFailed THEN
			CheckTrackTable := -1;
		 	      sInfoText := 'End at track implausible!';	
		ELSIF bTrackTablePlausible THEN
			CheckTrackTable := 1;
		 	      sInfoText := 'TrackTable check successful';
		ELSE
			CheckTrackTable := -UINT_TO_DINT(nTableImplausibleIndex);
			      sInfoText := CONCAT('TrackTable check failed at track point: ', UINT_TO_STRING(nTableImplausibleIndex));
		END_IF

		nStateCheckTabel := 0;
		
	END_CASE
END_METHOD

METHOD ClearTrackTable : BOOL
VAR_INPUT
END_VAR


	bStartingTrackFailed := FALSE;
	bEndingTrackFailed	 := FALSE;
	
	
	nTrackTableIndex := 0;
	MEMSET(ADR(TrackTable),0,SIZEOF(TrackTable));
	MEMSET(ADR(stTrackBuildParameter),0,SIZEOF(stTrackBuildParameter));
	
	
	sInfoText := 'TrackTable cleared';
	
	ClearTrackTable := TRUE;
END_METHOD

PROPERTY P_BuildlParameter : ST_TrackBuildParameter
GET
	P_BuildlParameter := stTrackBuildParameter;
END_GET
END_PROPERTY

PROPERTY P_CloseTheLoop : BOOL
GET
P_CloseTheLoop := bCloseTheLoop;
END_GET
SET
bCloseTheLoop := P_CloseTheLoop;

IF bCloseTheLoop THEN
	sInfoText := 'Set CloseTheLoop';
ELSE
	sInfoText := 'Cleared CloseTheLoop';
END_IF
END_SET
END_PROPERTY

PROPERTY P_EndAtTrack : I_TrackStandard
GET
	P_EndAtTrack := stTrackBuildParameter.EndAtTrack;
END_GET
SET
IF P_EndAtTrack <> 0 THEN
	IF P_EndAtTrack.ref <> 0 THEN
	      stTrackBuildParameter.EndAtTrack := P_EndAtTrack;
		  
		  bEndingTrackFailed := FALSE;
		           sInfoText := 'Added ending track successfully';
	ELSE
		bEndingTrackFailed := TRUE;
		sInfoText := 'Adding failed, object reference is null!';
	END_IF
ELSE
	bEndingTrackFailed := TRUE;
	sInfoText := 'Adding failed, object is null!';
END_IF
END_SET
END_PROPERTY

PROPERTY P_InfoText : STRING
GET


	P_InfoText := sInfoText;
END_GET
END_PROPERTY

PROPERTY P_NumberOfPointsInTable : UINT
GET
	

	P_NumberOfPointsInTable := nTrackTableIndex;
END_GET
END_PROPERTY

PROPERTY P_StartFromTrack : I_TrackStandard
GET
	P_StartFromTrack := stTrackBuildParameter.StartFromTrack;
END_GET
SET
IF P_StartFromTrack <> 0 THEN
	IF P_StartFromTrack.ref <> 0 THEN
		stTrackBuildParameter.StartFromTrack := P_StartFromTrack;
		
		bStartingTrackFailed := FALSE;
		           sInfoText := 'Added starting track successfully';
	ELSE
		bStartingTrackFailed := TRUE;
		sInfoText := 'Adding failed, object reference is null!';
	END_IF
ELSE
	bStartingTrackFailed := TRUE;
	sInfoText := 'Adding failed, object is null!';
END_IF
END_SET
END_PROPERTY

PROPERTY P_Table : REFERENCE TO ARRAY[1..maxNumTrackPoints] OF ST_TrackTable
GET
P_Table REF= TrackTable;
END_GET
END_PROPERTY

PROPERTY P_TrackCheckImplausibleTableIndex : UINT
GET
P_TrackCheckImplausibleTableIndex := nTableImplausibleIndex;
END_GET
END_PROPERTY

PROPERTY P_TrackTableCheckResult : BOOL
GET
P_TrackTableCheckResult := bTrackTablePlausible;
END_GET
END_PROPERTY

END_FUNCTION_BLOCK

// XPlanarStandardFunctions/MotionSystem/FB_XPlanarSystem
FUNCTION_BLOCK FB_XPlanarSystem  IMPLEMENTS I_MotionSystem

VAR_OUTPUT
END_VAR
VAR
	// Utility
	nIndexXPU				: UINT;
	nStateInitXpu			: INT;
	sInitInfo				: STRING :='not called';
	bSystemInitialized		: BOOL;	
	
	{attribute 'hide'}
	ipXpuInternal			: I_TcIoXPlanarProcessingUnit;	
	{attribute 'hide'}
	ipTcIoXPlanarMover		: ARRAY [1..Params_XPlanar.maxNumMover] OF I_TcIoXPlanarMover;
	{attribute 'hide'}
	ipTcIoXPlanarTile		: ARRAY [1..Param_TcIoXplanarEnvironment.MaxTiles] OF I_TcIoXPlanarTile;

	

	// XPlanar components
	ipMover 				: ARRAY [1..Params_XPlanar.maxNumMover] OF I_XPlanarMoverStandard;	
	ipTrack					: ARRAY [1..Params_XPlanar.maxTrackCount] OF I_TrackStandard;
	
	environment				: MC_PlanarEnvironment;
	group					: MC_PlanarGroup;
	part					: ARRAY [1..Params_XPlanar.maxNumberOfParts] OF MC_PlanarPart;
	
	
	
	
	{attribute 'hide'}
	_nAxisCount				: INT;
	{attribute 'hide'}	
	_nTrackCount			: INT;
	{attribute 'hide'}
	eState 					: E_MethodKeepAliveMotionSystem;
	{attribute 'hide'}	
	nState					: INT;
	
	
	// Return Properties
	stRtAddMover			: ST_CommandReturn;
	stRtAddMovers			: ST_CommandReturn;
	stRtDisableGroup		: ST_CommandReturn;
	stRtDisableMovers		: ST_CommandReturn;
	stRtDisableSystem		: ST_CommandReturn;
	stRtEnableGroup			: ST_CommandReturn;
	stRtEnableMovers		: ST_CommandReturn;
	stRtEnableSystem		: ST_CommandReturn;
	stRtHaltSystem			: ST_CommandReturn;
	stRtLeaveTrack			: ST_CommandReturn;
	stRtRemoveMover			: ST_CommandReturn;
	stRtResetGroup			: ST_CommandReturn;
	stRtRemoveMovers		: ST_CommandReturn;
	stRtResetMovers			: ST_CommandReturn;
	stRtResetTracks			: ST_CommandReturn;
	stRtResetSystem			: ST_CommandReturn;
	stRtAddEnvironment		: ST_CommandReturn;
	stRtRemoveEnvironment	: ST_CommandReturn;	
	stRtAddTracks			: ST_CommandReturn;
	stRtRemoveTracks		: ST_CommandReturn;
	stRtEnableTrack			: ST_CommandReturn;
	stRtEnableTracks		: ST_CommandReturn;	
	stRtDisableTracks		: ST_CommandReturn;	
	stRtAddModule			: ST_CommandReturn;
	stRtPartInitialize			: ST_CommandReturn;
	stRtPartInitializeMulti		: ST_CommandReturn;
	stRtPartActivatePosition	: ST_CommandReturn;
	stRtPartForceDisable		: ST_CommandReturn;	
	stRtPartForceEnable			: ST_CommandReturn;	
	stRtPartAllowEnable			: ST_CommandReturn;		
	stRtPartReset				: ST_CommandReturn;	
	stRtResetParts				: ST_CommandReturn;	
	
	{attribute 'hide'}
	stValidMoverCheckInfo	: ST_MoverCheckInfo;
	
	// addModuleToEnvironment
	{attribute 'hide'}	
	_addModulePositionX : LREAL;
	{attribute 'hide'}	
	_addModulePositionY : LREAL;
	
	// Add/Remove Mover to/from Group
	{attribute 'hide'}
	MoverToAdd 				: I_XPlanarMoverStandard;
	{attribute 'hide'}
	MoverToRemove			: I_XPlanarMoverStandard;
	
	// Enable a single track
	{attribute 'hide'}
	TrackToEnable			: I_TrackStandard;
	
	
	{attribute 'hide'}
	PartToInitialze			: OTCID;	
	{attribute 'hide'}
	PartToDisable			: UDINT;
	{attribute 'hide'}
	PartToEnableAllow		: UDINT;
	{attribute 'hide'}
	PartToEnableForce		: UDINT;		
	{attribute 'hide'}
	PartToReset				: UDINT;
	{attribute 'hide'}
	AddressArrayPartID		: PVOID;
	{attribute 'hide'}
	nPartCnt				: UINT;	
	{attribute 'hide'}
	nPartActivateIndex		: UINT;
	{attribute 'hide'}
	nPositionActivateIndex	: UINT;	
	
	
	
	
	//******
	{attribute 'hide'}
	nForCounter 			: DINT;
	{attribute 'hide'}
	idx						: UDINT;
	{attribute 'hide'}
	cmdFeedback				: MC_PlanarFeedback;
	{attribute 'hide'}
	bDone 					: BOOL;
	{attribute 'hide'}
	bError					: BOOL;
	{attribute 'hide'}
	nErrorID				: UDINT;
	{attribute 'hide'}
	stResultErrorInfo		: ST_CommandReturnInfo;	
	{attribute 'hide'}
	_bResultDone			: BOOL;
	{attribute 'hide'}
	_bResultError			: BOOL;
	{attribute 'hide'}
	_nResultErrorID			: UDINT;
	{attribute 'hide'}
	_stResultErrorInfo		: ST_CommandReturnInfo;
	{attribute 'hide'}
	_stResultErrorInfoClear	: ST_CommandReturnInfo;
	
	
	{attribute 'hide'}
	fbMsg : FB_TcMessage; 
	{attribute 'hide'}
	bInit : BOOL := TRUE;
	{attribute 'hide'} 
    bSend : BOOL := TRUE; 
	
	
	
	
END_VAR

PROPERTY P_AddEnviromentToGroup : REFERENCE TO ST_CommandReturn
GET
P_AddEnviromentToGroup REF= stRtAddEnvironment;
END_GET
END_PROPERTY

PROPERTY P_AddModuleToEnvironment : REFERENCE TO ST_CommandReturn
GET
P_AddModuleToEnvironment REF= stRtAddModule;
END_GET
END_PROPERTY

PROPERTY P_AddMoversToGroup : REFERENCE TO ST_CommandReturn
GET
P_AddMoversToGroup REF= stRtAddMovers;
END_GET
END_PROPERTY

PROPERTY P_AddMoverToGroup : REFERENCE TO ST_CommandReturn
GET
P_AddMoverToGroup REF= stRtAddMover;
END_GET
END_PROPERTY

PROPERTY P_AddTracksToGroup : REFERENCE TO ST_CommandReturn
GET
P_AddTracksToGroup REF= stRtAddTracks;
END_GET
END_PROPERTY

PROPERTY P_CheckValidMovers : REFERENCE TO ST_MoverCheckInfo
GET
P_CheckValidMovers Ref= stValidMoverCheckInfo;
END_GET
END_PROPERTY

PROPERTY P_DisableGroup : REFERENCE TO ST_CommandReturn
GET
P_DisableGroup REF= stRtDisableGroup;
END_GET
END_PROPERTY

PROPERTY P_DisableMovers : REFERENCE TO ST_CommandReturn
GET
P_DisableMovers REF= stRtDisableMovers;
END_GET
END_PROPERTY

PROPERTY P_DisableTracks : REFERENCE TO ST_CommandReturn
GET
P_DisableTracks REF= stRtDisableTracks;
END_GET
END_PROPERTY

PROPERTY P_EnableGroup : REFERENCE TO ST_CommandReturn
GET
P_EnableGroup REF= stRtEnableGroup;
END_GET
END_PROPERTY

PROPERTY P_EnableMovers : REFERENCE TO ST_CommandReturn
GET
P_EnableMovers REF= stRtEnableMovers;
END_GET
END_PROPERTY

PROPERTY P_EnableTrack : REFERENCE TO ST_CommandReturn
GET
P_EnableTrack REF= stRtEnableTrack;
END_GET
END_PROPERTY

PROPERTY P_EnableTracks : REFERENCE TO ST_CommandReturn
GET
P_EnableTracks REF= stRtEnableTracks;
END_GET
END_PROPERTY

PROPERTY P_HaltSystem : REFERENCE TO ST_CommandReturn
GET
P_HaltSystem REF= stRtHaltSystem;
END_GET
END_PROPERTY

PROPERTY P_LeaveTrack : REFERENCE TO ST_CommandReturn
GET
P_LeaveTrack REF= stRtLeaveTrack;
END_GET
END_PROPERTY

PROPERTY P_PartActivatePosition : REFERENCE TO ST_CommandReturn
GET
P_PartActivatePosition REF= stRtPartActivatePosition;
END_GET
END_PROPERTY

PROPERTY P_PartAllowEnable : REFERENCE TO ST_CommandReturn
GET
P_PartAllowEnable REF= stRtPartAllowEnable;
END_GET
END_PROPERTY

PROPERTY P_PartForceDisable : REFERENCE TO ST_CommandReturn
GET
P_PartForceDisable REF= stRtPartForceDisable;
END_GET
END_PROPERTY

PROPERTY P_PartForceEnable : REFERENCE TO ST_CommandReturn
GET
P_PartForceEnable REF= stRtPartForceEnable;
END_GET
END_PROPERTY

PROPERTY P_PartInitialize : REFERENCE TO ST_CommandReturn
GET
P_PartInitialize REF= stRtPartInitialize;
END_GET
END_PROPERTY

PROPERTY P_PartInitializeMulti : REFERENCE TO ST_CommandReturn
GET
P_PartInitializeMulti REF= stRtPartInitializeMulti;
END_GET
END_PROPERTY

PROPERTY P_PartReset : REFERENCE TO ST_CommandReturn
GET
P_PartReset REF= stRtPartReset;
END_GET
END_PROPERTY

PROPERTY P_RemoveEnviromentFromGroup : REFERENCE TO ST_CommandReturn
GET
P_RemoveEnviromentFromGroup REF= stRtRemoveEnvironment;
END_GET
END_PROPERTY

PROPERTY P_RemoveMoverFromGroup : REFERENCE TO ST_CommandReturn
GET
P_RemoveMoverFromGroup REF= stRtRemoveMover;
END_GET
END_PROPERTY

PROPERTY P_RemoveMoversFromGroup : REFERENCE TO ST_CommandReturn
GET
P_RemoveMoversFromGroup REF= stRtRemoveMovers;
END_GET
END_PROPERTY

PROPERTY P_RemoveTracksFromGroup : REFERENCE TO ST_CommandReturn
GET
P_RemoveTracksFromGroup REF= stRtRemoveTracks;
END_GET
END_PROPERTY

PROPERTY P_ResetGroup : REFERENCE TO ST_CommandReturn
GET
P_ResetGroup REF= stRtResetGroup;
END_GET
END_PROPERTY

PROPERTY P_ResetMovers : REFERENCE TO ST_CommandReturn
GET
P_ResetMovers REF= stRtResetMovers;
END_GET
END_PROPERTY

PROPERTY P_ResetParts : REFERENCE TO ST_CommandReturn
GET
P_ResetParts REF= stRtResetParts;
END_GET
END_PROPERTY

PROPERTY P_ResetTracks : REFERENCE TO ST_CommandReturn
GET
P_ResetTracks REF= stRtResetTracks;
END_GET
END_PROPERTY

METHOD AddEnvironmentToGroup : BOOL
IF eState = E_MethodKeepAliveMotionSystem.eIdle THEN
	MEMSET(ADR(stRtAddEnvironment), 0, SIZEOF(stRtAddEnvironment));
	eState := E_MethodKeepAliveMotionSystem.eAddEnvironmentToGroup;
	AddEnvironmentToGroup := TRUE;
ELSE
	AddEnvironmentToGroup := FALSE;
END_IF
END_METHOD

METHOD AddModuleToEnvironment : BOOL
VAR_INPUT
	xPos : LREAL;
	yPos : LREAL;
END_VAR
IF eState = E_MethodKeepAliveMotionSystem.eIdle THEN
	MEMSET(ADR(stRtAddModule), 0, SIZEOF(stRtAddModule));
	_addModulePositionX := xPos;
	_addModulePositionY := yPos;
 	eState := E_MethodKeepAliveMotionSystem.eAddModuleToEnvironment;
	AddModuleToEnvironment := TRUE;
ELSE
	AddModuleToEnvironment := FALSE;
END_IF
END_METHOD

METHOD AddMoversToGroup : BOOL
IF eState = E_MethodKeepAliveMotionSystem.eIdle THEN
	MEMSET(ADR(stRtAddMovers), 0, SIZEOF(stRtAddMovers));
	eState := E_MethodKeepAliveMotionSystem.eAddMoversToGroup;
	AddMoversToGroup := TRUE;
ELSE
	AddMoversToGroup := FALSE;
END_IF
END_METHOD

METHOD AddMoverToGroup : BOOL
VAR_INPUT
	ipMover		: I_XPlanarMoverStandard;
END_VAR
IF eState = E_MethodKeepAliveMotionSystem.eIdle THEN
	MEMSET(ADR(stRtAddMover), 0, SIZEOF(stRtAddMover));
	         eState := E_MethodKeepAliveMotionSystem.eAddMoverToGroup;
	     MoverToAdd := ipMover;
	AddMoverToGroup := TRUE;
ELSE
	AddMoverToGroup := FALSE;
END_IF
END_METHOD

METHOD AddTracksToGroup : BOOL


VAR_INST
	nTestCounter01 : UINT;	
	
END_VAR
IF eState = E_MethodKeepAliveMotionSystem.eIdle THEN
	MEMSET(ADR(stRtAddTracks), 0, SIZEOF(stRtAddTracks));
	eState := E_MethodKeepAliveMotionSystem.eAddTracksToGroup;
	AddTracksToGroup := TRUE;
	
	nTestCounter01 := nTestCounter01 +1;
ELSE
	AddTracksToGroup := FALSE;
END_IF
END_METHOD

METHOD CheckValidMovers : BOOL
VAR_INPUT
END_VAR
IF eState = E_MethodKeepAliveMotionSystem.eIdle THEN
	IF bSystemInitialized THEN	
		MEMSET(ADR(stValidMoverCheckInfo), 0, SIZEOF(stValidMoverCheckInfo));
		eState := E_MethodKeepAliveMotionSystem.eCheckValidMovers;
		CheckValidMovers := TRUE;
	END_IF
ELSE
	CheckValidMovers := FALSE;
END_IF
END_METHOD

METHOD DisableGroup : BOOL
IF eState = E_MethodKeepAliveMotionSystem.eIdle THEN
	MEMSET(ADR(stRtDisableGroup), 0, SIZEOF(stRtDisableGroup));
	eState := E_MethodKeepAliveMotionSystem.eDisableGroup;
	DisableGroup := TRUE;
ELSE
	DisableGroup := FALSE;
END_IF
END_METHOD

METHOD DisableMovers : BOOL
ResetStateVariables();
MEMSET(ADR(stRtDisableMovers), 0, SIZEOF(stRtDisableMovers));
eState := E_MethodKeepAliveMotionSystem.eDisableMovers;
DisableMovers := TRUE;
END_METHOD

METHOD DisableTracks : BOOL
VAR_INPUT
END_VAR
IF eState = E_MethodKeepAliveMotionSystem.eIdle THEN
	MEMSET(ADR(stRtDisableTracks), 0, SIZEOF(stRtDisableTracks));
	eState := E_MethodKeepAliveMotionSystem.eDisableTracks;
	DisableTracks := TRUE;
ELSE
	DisableTracks := FALSE;
END_IF
END_METHOD

METHOD EnableGroup : BOOL
IF eState = E_MethodKeepAliveMotionSystem.eIdle THEN
	MEMSET(ADR(stRtEnableGroup), 0, SIZEOF(stRtEnableGroup));
	eState := E_MethodKeepAliveMotionSystem.eEnableGroup;
	EnableGroup := TRUE;
ELSE
	EnableGroup := FALSE;
END_IF
END_METHOD

METHOD EnableMovers : BOOL
IF eState = E_MethodKeepAliveMotionSystem.eIdle THEN
	MEMSET(ADR(stRtEnableMovers), 0, SIZEOF(stRtEnableMovers));
	eState := E_MethodKeepAliveMotionSystem.eEnableMovers;
	EnableMovers := TRUE;
ELSE
	EnableMovers := FALSE;
END_IF
END_METHOD

METHOD EnableTrack : BOOL
VAR_INPUT
	ipTrackToAdd	: I_TrackStandard;
END_VAR
IF eState = E_MethodKeepAliveMotionSystem.eIdle THEN
	MEMSET(ADR(stRtEnableTrack), 0, SIZEOF(stRtEnableTrack));
	TrackToEnable := ipTrackToAdd;
	       eState := E_MethodKeepAliveMotionSystem.eEnableTrack;
	  EnableTrack := TRUE;
ELSE
	EnableTrack := FALSE;
END_IF
END_METHOD

METHOD EnableTracks : BOOL
VAR_INPUT
END_VAR
IF eState = E_MethodKeepAliveMotionSystem.eIdle THEN
	MEMSET(ADR(stRtEnableTracks), 0, SIZEOF(stRtEnableTracks));
	eState := E_MethodKeepAliveMotionSystem.eEnableTracks;
	EnableTracks := TRUE;
ELSE
	EnableTracks := FALSE;
END_IF
END_METHOD

METHOD HaltSystem : BOOL
IF eState = E_MethodKeepAliveMotionSystem.eIdle THEN
	MEMSET(ADR(stRtHaltSystem), 0, SIZEOF(stRtHaltSystem));
	eState := E_MethodKeepAliveMotionSystem.eHaltSystem;
	HaltSystem := TRUE;
ELSE
	HaltSystem := FALSE;
END_IF
END_METHOD

METHOD LeaveTrack : BOOL
IF eState = E_MethodKeepAliveMotionSystem.eIdle THEN
	MEMSET(ADR(stRtLeaveTrack), 0, SIZEOF(stRtLeaveTrack));
	eState := E_MethodKeepAliveMotionSystem.eLeaveTrack;
	LeaveTrack := TRUE;
ELSE
	LeaveTrack := FALSE;
END_IF
END_METHOD

METHOD PartActivatePosition : BOOL
VAR_INPUT
	nPartIndex		: UINT;
	nPositionIndex	: UINT;
END_VAR

